Yaskawa INFORM job: A_ROOF_UPPER_0614_2_PAINT_34.JBI

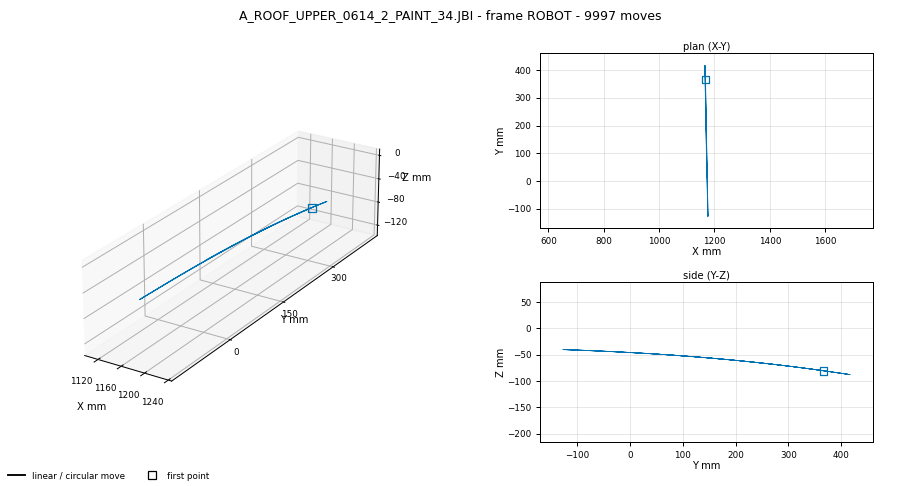
[picture p0: tool path of A_ROOF_UPPER_0614_2_PAINT_34.JBI in frame ROBOT, 9997 of 9997 moves have a stored position in this frame; points joined in program order, loops and branches not executed]
/JOB
//NAME A_ROOF_UPPER_0614_2_PAINT34
//POS
///NPOS 9997,0,0,0,0,0
///TOOL 1
///USER 0
///POSTYPE ROBOT
///RECTAN
///RCONF 1,0,0,0,0,0,0,0,0,0,0,0,0,0,0,0,0,0,0,0,0,0,0,0
C00000=1167.748,366.812,-80.185,-176.180,8.924,148.683
C00001=1167.752,366.565,-80.149,-176.183,8.920,148.683
C00002=1167.756,366.317,-80.115,-176.185,8.916,148.683
C00003=1167.761,366.035,-80.075,-176.187,8.912,148.682
C00004=1167.765,365.752,-80.035,-176.190,8.907,148.682
C00005=1167.770,365.471,-79.996,-176.191,8.904,148.681
C00006=1167.774,365.188,-79.956,-176.194,8.899,148.681
C00007=1167.778,364.940,-79.921,-176.196,8.895,148.680
C00008=1167.782,364.693,-79.887,-176.199,8.892,148.680
C00009=1167.786,364.446,-79.851,-176.200,8.888,148.680
C00010=1167.790,364.198,-79.817,-176.203,8.884,148.679
C00011=1167.794,363.950,-79.782,-176.205,8.880,148.679
C00012=1167.797,363.703,-79.747,-176.207,8.877,148.679
C00013=1167.802,363.456,-79.713,-176.209,8.872,148.678
C00014=1167.806,363.207,-79.678,-176.212,8.869,148.678
C00015=1167.809,362.960,-79.644,-176.214,8.865,148.677
C00016=1167.813,362.713,-79.608,-176.216,8.861,148.677
C00017=1167.818,362.465,-79.574,-176.218,8.858,148.677
C00018=1167.821,362.218,-79.540,-176.220,8.854,148.676
C00019=1167.825,361.970,-79.505,-176.223,8.850,148.676
C00020=1167.829,361.722,-79.470,-176.225,8.846,148.676
C00021=1167.833,361.475,-79.437,-176.227,8.843,148.675
C00022=1167.837,361.227,-79.402,-176.230,8.839,148.675
C00023=1167.842,360.980,-79.367,-176.232,8.835,148.675
C00024=1167.845,360.732,-79.332,-176.234,8.832,148.674
C00025=1167.849,360.485,-79.298,-176.237,8.828,148.674
C00026=1167.853,360.237,-79.263,-176.239,8.824,148.674
C00027=1167.857,359.990,-79.229,-176.241,8.820,148.673
C00028=1167.862,359.742,-79.195,-176.244,8.817,148.673
C00029=1167.865,359.494,-79.160,-176.245,8.813,148.673
C00030=1167.869,359.247,-79.126,-176.248,8.809,148.672
C00031=1167.873,358.999,-79.091,-176.251,8.806,148.672
C00032=1167.877,358.752,-79.057,-176.252,8.802,148.672
C00033=1167.881,358.504,-79.022,-176.255,8.798,148.671
C00034=1167.885,358.256,-78.989,-176.258,8.795,148.671
C00035=1167.890,358.009,-78.954,-176.259,8.791,148.671
C00036=1167.893,357.761,-78.920,-176.262,8.787,148.671
C00037=1167.897,357.514,-78.885,-176.265,8.784,148.670
C00038=1167.901,357.265,-78.852,-176.266,8.780,148.670
C00039=1167.906,357.018,-78.817,-176.269,8.776,148.670
C00040=1167.909,356.771,-78.784,-176.272,8.773,148.669
C00041=1167.913,356.523,-78.749,-176.274,8.769,148.669
C00042=1167.917,356.276,-78.715,-176.276,8.765,148.669
C00043=1167.921,356.027,-78.680,-176.279,8.762,148.669
C00044=1167.925,355.780,-78.646,-176.281,8.758,148.668
C00045=1167.930,355.532,-78.612,-176.283,8.754,148.668
C00046=1167.933,355.285,-78.578,-176.286,8.750,148.668
C00047=1167.938,355.037,-78.544,-176.288,8.747,148.667
C00048=1167.942,354.790,-78.510,-176.291,8.743,148.667
C00049=1167.945,354.542,-78.476,-176.293,8.739,148.667
C00050=1167.950,354.294,-78.442,-176.295,8.736,148.666
C00051=1167.953,354.047,-78.408,-176.298,8.732,148.666
C00052=1167.957,353.799,-78.373,-176.300,8.729,148.666
C00053=1167.962,353.551,-78.340,-176.302,8.725,148.666
C00054=1167.965,353.304,-78.306,-176.305,8.721,148.665
C00055=1167.969,353.056,-78.271,-176.307,8.718,148.665
C00056=1167.974,352.808,-78.238,-176.309,8.714,148.665
C00057=1167.978,352.561,-78.204,-176.312,8.711,148.665
C00058=1167.982,352.312,-78.170,-176.315,8.707,148.664
C00059=1167.985,352.065,-78.136,-176.316,8.703,148.664
C00060=1167.990,351.818,-78.102,-176.319,8.700,148.664
C00061=1167.994,351.570,-78.069,-176.322,8.696,148.664
C00062=1167.997,351.322,-78.034,-176.324,8.693,148.663
C00063=1168.002,351.074,-78.001,-176.326,8.689,148.663
C00064=1168.006,350.827,-77.967,-176.329,8.685,148.663
C00065=1168.010,350.579,-77.934,-176.331,8.682,148.662
C00066=1168.013,350.332,-77.899,-176.333,8.678,148.662
C00067=1168.018,350.084,-77.866,-176.335,8.675,148.662
C00068=1168.022,349.836,-77.832,-176.338,8.671,148.662
C00069=1168.026,349.589,-77.799,-176.341,8.668,148.661
C00070=1168.030,349.341,-77.764,-176.343,8.664,148.661
C00071=1168.034,349.093,-77.731,-176.346,8.660,148.661
C00072=1168.038,348.846,-77.697,-176.348,8.657,148.661
C00073=1168.042,348.598,-77.664,-176.350,8.654,148.661
C00074=1168.047,348.350,-77.630,-176.352,8.650,148.660
C00075=1168.050,348.102,-77.596,-176.355,8.646,148.660
C00076=1168.055,347.854,-77.562,-176.357,8.643,148.660
C00077=1168.059,347.607,-77.529,-176.360,8.639,148.659
C00078=1168.063,347.360,-77.495,-176.362,8.636,148.659
C00079=1168.067,347.112,-77.462,-176.365,8.632,148.659
C00080=1168.070,346.863,-77.429,-176.367,8.629,148.659
C00081=1168.075,346.616,-77.394,-176.369,8.625,148.659
C00082=1168.079,346.368,-77.361,-176.372,8.622,148.658
C00083=1168.083,346.121,-77.328,-176.374,8.618,148.658
C00084=1168.087,345.873,-77.294,-176.377,8.615,148.658
C00085=1168.091,345.626,-77.261,-176.379,8.611,148.658
C00086=1168.095,345.378,-77.228,-176.381,8.608,148.657
C00087=1168.099,345.130,-77.194,-176.384,8.604,148.657
C00088=1168.104,344.882,-77.161,-176.386,8.601,148.657
C00089=1168.107,344.634,-77.127,-176.389,8.597,148.657
C00090=1168.112,344.387,-77.093,-176.391,8.594,148.657
C00091=1168.116,344.139,-77.060,-176.394,8.590,148.656
C00092=1168.120,343.891,-77.027,-176.396,8.587,148.656
C00093=1168.124,343.644,-76.994,-176.398,8.583,148.656
C00094=1168.128,343.396,-76.961,-176.401,8.580,148.656
C00095=1168.132,343.148,-76.928,-176.404,8.576,148.655
C00096=1168.136,342.900,-76.895,-176.406,8.573,148.655
C00097=1168.140,342.653,-76.860,-176.408,8.569,148.655
C00098=1168.144,342.405,-76.827,-176.410,8.566,148.655
C00099=1168.148,342.157,-76.794,-176.413,8.562,148.655
C00100=1168.152,341.909,-76.761,-176.416,8.559,148.654
C00101=1168.156,341.662,-76.728,-176.418,8.555,148.654
C00102=1168.160,341.414,-76.695,-176.420,8.552,148.654
C00103=1168.164,341.166,-76.661,-176.423,8.549,148.654
C00104=1168.169,340.918,-76.628,-176.425,8.545,148.653
C00105=1168.173,340.671,-76.595,-176.428,8.542,148.653
C00106=1168.177,340.423,-76.562,-176.430,8.538,148.653
C00107=1168.182,340.143,-76.525,-176.433,8.534,148.653
C00108=1168.186,339.863,-76.488,-176.436,8.530,148.653
C00109=1168.191,339.585,-76.451,-176.438,8.527,148.652
C00110=1168.195,339.305,-76.413,-176.441,8.523,148.652
C00111=1168.200,339.057,-76.380,-176.444,8.519,148.652
C00112=1168.204,338.810,-76.347,-176.446,8.515,148.652
C00113=1168.208,338.562,-76.314,-176.449,8.512,148.652
C00114=1168.212,338.314,-76.281,-176.451,8.509,148.652
C00115=1168.216,338.066,-76.248,-176.454,8.506,148.651
C00116=1168.220,337.818,-76.216,-176.456,8.502,148.651
C00117=1168.224,337.571,-76.183,-176.459,8.498,148.651
C00118=1168.228,337.323,-76.150,-176.461,8.495,148.651
C00119=1168.232,337.075,-76.116,-176.463,8.492,148.650
C00120=1168.237,336.827,-76.084,-176.466,8.488,148.650
C00121=1168.240,336.579,-76.051,-176.468,8.485,148.650
C00122=1168.244,336.332,-76.018,-176.471,8.482,148.650
C00123=1168.249,336.083,-75.986,-176.474,8.478,148.650
C00124=1168.253,335.836,-75.953,-176.476,8.475,148.650
C00125=1168.257,335.588,-75.919,-176.478,8.471,148.649
C00126=1168.261,335.340,-75.888,-176.480,8.468,148.649
C00127=1168.265,335.092,-75.854,-176.483,8.465,148.649
C00128=1168.269,334.844,-75.821,-176.486,8.461,148.649
C00129=1168.273,334.596,-75.789,-176.488,8.458,148.649
C00130=1168.277,334.349,-75.756,-176.491,8.454,148.649
C00131=1168.282,334.102,-75.724,-176.493,8.451,148.648
C00132=1168.286,333.853,-75.691,-176.496,8.448,148.648
C00133=1168.289,333.606,-75.659,-176.498,8.445,148.648
C00134=1168.294,333.357,-75.626,-176.501,8.441,148.648
C00135=1168.298,333.110,-75.593,-176.503,8.437,148.648
C00136=1168.302,332.862,-75.561,-176.506,8.434,148.648
C00137=1168.306,332.614,-75.528,-176.508,8.431,148.647
C00138=1168.310,332.366,-75.495,-176.510,8.428,148.647
C00139=1168.314,332.118,-75.463,-176.513,8.424,148.647
C00140=1168.319,331.871,-75.431,-176.516,8.420,148.647
C00141=1168.323,331.623,-75.398,-176.518,8.417,148.647
C00142=1168.327,331.375,-75.366,-176.521,8.414,148.647
C00143=1168.331,331.127,-75.333,-176.523,8.411,148.646
C00144=1168.334,330.879,-75.301,-176.525,8.408,148.646
C00145=1168.339,330.631,-75.268,-176.528,8.405,148.646
C00146=1168.344,330.384,-75.236,-176.531,8.400,148.646
C00147=1168.347,330.136,-75.204,-176.533,8.397,148.646
C00148=1168.351,329.888,-75.171,-176.536,8.394,148.646
C00149=1168.355,329.640,-75.139,-176.538,8.391,148.646
C00150=1168.360,329.391,-75.106,-176.540,8.388,148.645
C00151=1168.364,329.144,-75.073,-176.543,8.384,148.645
C00152=1168.368,328.896,-75.042,-176.546,8.380,148.645
C00153=1168.372,328.648,-75.009,-176.548,8.377,148.645
C00154=1168.376,328.401,-74.977,-176.550,8.374,148.645
C00155=1168.380,328.152,-74.944,-176.553,8.371,148.645
C00156=1168.385,327.905,-74.913,-176.556,8.368,148.645
C00157=1168.389,327.657,-74.880,-176.558,8.364,148.644
C00158=1168.392,327.409,-74.848,-176.560,8.361,148.644
C00159=1168.397,327.161,-74.815,-176.563,8.357,148.644
C00160=1168.401,326.913,-74.783,-176.566,8.354,148.644
C00161=1168.405,326.665,-74.752,-176.568,8.351,148.644
C00162=1168.409,326.417,-74.720,-176.571,8.348,148.644
C00163=1168.413,326.170,-74.687,-176.573,8.344,148.643
C00164=1168.417,325.921,-74.655,-176.575,8.341,148.643
C00165=1168.422,325.674,-74.623,-176.578,8.338,148.643
C00166=1168.426,325.426,-74.591,-176.580,8.335,148.643
C00167=1168.430,325.178,-74.559,-176.583,8.331,148.643
C00168=1168.434,324.930,-74.527,-176.586,8.328,148.643
C00169=1168.438,324.682,-74.495,-176.588,8.324,148.643
C00170=1168.442,324.434,-74.463,-176.590,8.321,148.642
C00171=1168.447,324.186,-74.431,-176.593,8.318,148.642
C00172=1168.451,323.938,-74.399,-176.595,8.315,148.642
C00173=1168.455,323.690,-74.367,-176.598,8.312,148.642
C00174=1168.459,323.442,-74.335,-176.601,8.309,148.642
C00175=1168.463,323.194,-74.303,-176.603,8.304,148.642
C00176=1168.467,322.946,-74.272,-176.606,8.301,148.642
C00177=1168.471,322.698,-74.240,-176.608,8.298,148.642
C00178=1168.476,322.451,-74.208,-176.611,8.295,148.641
C00179=1168.479,322.203,-74.176,-176.613,8.292,148.641
C00180=1168.483,321.955,-74.144,-176.616,8.289,148.641
C00181=1168.488,321.707,-74.112,-176.618,8.286,148.641
C00182=1168.492,321.459,-74.080,-176.621,8.282,148.641
C00183=1168.496,321.211,-74.048,-176.623,8.279,148.641
C00184=1168.500,320.964,-74.017,-176.626,8.275,148.641
C00185=1168.504,320.715,-73.984,-176.629,8.272,148.641
C00186=1168.508,320.467,-73.952,-176.631,8.269,148.641
C00187=1168.513,320.219,-73.922,-176.634,8.266,148.640
C00188=1168.516,319.971,-73.890,-176.636,8.262,148.640
C00189=1168.521,319.724,-73.858,-176.639,8.259,148.640
C00190=1168.525,319.476,-73.826,-176.641,8.256,148.640
C00191=1168.529,319.227,-73.794,-176.644,8.253,148.640
C00192=1168.534,318.980,-73.763,-176.646,8.250,148.640
C00193=1168.537,318.731,-73.731,-176.649,8.247,148.640
C00194=1168.542,318.484,-73.700,-176.651,8.244,148.640
C00195=1168.546,318.236,-73.667,-176.654,8.239,148.639
C00196=1168.550,317.987,-73.636,-176.657,8.236,148.639
C00197=1168.554,317.740,-73.605,-176.659,8.233,148.639
C00198=1168.558,317.492,-73.573,-176.662,8.230,148.639
C00199=1168.563,317.244,-73.542,-176.664,8.227,148.639
C00200=1168.566,316.996,-73.510,-176.667,8.224,148.639
C00201=1168.571,316.748,-73.479,-176.669,8.221,148.639
C00202=1168.575,316.500,-73.448,-176.672,8.218,148.639
C00203=1168.580,316.252,-73.416,-176.674,8.214,148.639
C00204=1168.583,316.004,-73.384,-176.677,8.211,148.639
C00205=1168.587,315.755,-73.353,-176.679,8.208,148.639
C00206=1168.592,315.508,-73.321,-176.681,8.205,148.638
C00207=1168.596,315.259,-73.290,-176.685,8.201,148.638
C00208=1168.600,315.012,-73.259,-176.687,8.198,148.638
C00209=1168.604,314.763,-73.228,-176.690,8.195,148.638
C00210=1168.608,314.516,-73.196,-176.692,8.191,148.638
C00211=1168.613,314.239,-73.161,-176.695,8.188,148.638
C00212=1168.618,313.962,-73.127,-176.697,8.184,148.638
C00213=1168.622,313.685,-73.091,-176.700,8.181,148.638
C00214=1168.627,313.408,-73.056,-176.704,8.177,148.638
C00215=1168.632,313.160,-73.025,-176.706,8.174,148.638
C00216=1168.635,312.912,-72.993,-176.709,8.171,148.638
C00217=1168.640,312.664,-72.963,-176.711,8.168,148.637
C00218=1168.644,312.416,-72.931,-176.714,8.165,148.637
C00219=1168.648,312.168,-72.900,-176.716,8.162,148.637
C00220=1168.652,311.919,-72.869,-176.719,8.159,148.637
C00221=1168.657,311.672,-72.837,-176.721,8.155,148.637
C00222=1168.661,311.424,-72.807,-176.724,8.152,148.637
C00223=1168.664,311.176,-72.776,-176.726,8.149,148.637
C00224=1168.669,310.928,-72.745,-176.729,8.146,148.637
C00225=1168.673,310.680,-72.714,-176.731,8.143,148.637
C00226=1168.677,310.432,-72.683,-176.734,8.139,148.637
C00227=1168.682,310.184,-72.651,-176.737,8.136,148.636
C00228=1168.686,309.936,-72.620,-176.739,8.133,148.636
C00229=1168.690,309.688,-72.589,-176.742,8.129,148.636
C00230=1168.694,309.439,-72.558,-176.744,8.126,148.636
C00231=1168.699,309.192,-72.527,-176.747,8.123,148.636
C00232=1168.702,308.944,-72.497,-176.749,8.120,148.636
C00233=1168.707,308.695,-72.465,-176.752,8.117,148.636
C00234=1168.711,308.447,-72.435,-176.754,8.114,148.636
C00235=1168.716,308.199,-72.404,-176.757,8.111,148.636
C00236=1168.719,307.951,-72.372,-176.759,8.108,148.636
C00237=1168.723,307.704,-72.342,-176.762,8.105,148.636
C00238=1168.727,307.455,-72.311,-176.764,8.101,148.636
C00239=1168.732,307.207,-72.280,-176.767,8.098,148.636
C00240=1168.737,306.959,-72.249,-176.770,8.095,148.636
C00241=1168.741,306.710,-72.218,-176.772,8.092,148.635
C00242=1168.744,306.463,-72.188,-176.775,8.089,148.636
C00243=1168.749,306.215,-72.157,-176.777,8.086,148.635
C00244=1168.754,305.967,-72.126,-176.780,8.083,148.635
C00245=1168.757,305.719,-72.095,-176.783,8.080,148.635
C00246=1168.761,305.471,-72.064,-176.785,8.077,148.635
C00247=1168.766,305.223,-72.034,-176.788,8.074,148.635
C00248=1168.770,304.975,-72.003,-176.790,8.070,148.635
C00249=1168.774,304.727,-71.972,-176.793,8.067,148.635
C00250=1168.778,304.479,-71.942,-176.795,8.064,148.635
C00251=1168.783,304.230,-71.911,-176.798,8.061,148.635
C00252=1168.787,303.982,-71.880,-176.800,8.058,148.635
C00253=1168.791,303.734,-71.850,-176.803,8.055,148.635
C00254=1168.796,303.486,-71.820,-176.806,8.052,148.635
C00255=1168.800,303.238,-71.788,-176.808,8.049,148.635
C00256=1168.804,302.990,-71.758,-176.811,8.046,148.635
C00257=1168.808,302.742,-71.727,-176.813,8.043,148.635
C00258=1168.813,302.494,-71.697,-176.816,8.039,148.634
C00259=1168.816,302.246,-71.666,-176.818,8.036,148.634
C00260=1168.821,301.997,-71.636,-176.821,8.033,148.634
C00261=1168.825,301.749,-71.606,-176.823,8.030,148.634
C00262=1168.830,301.501,-71.575,-176.826,8.027,148.634
C00263=1168.834,301.253,-71.544,-176.829,8.024,148.634
C00264=1168.837,301.005,-71.514,-176.831,8.021,148.634
C00265=1168.842,300.757,-71.484,-176.834,8.018,148.634
C00266=1168.846,300.509,-71.454,-176.837,8.015,148.634
C00267=1168.851,300.261,-71.423,-176.839,8.012,148.634
C00268=1168.855,300.013,-71.393,-176.842,8.009,148.634
C00269=1168.859,299.764,-71.362,-176.844,8.006,148.634
C00270=1168.863,299.516,-71.332,-176.847,8.002,148.634
C00271=1168.868,299.268,-71.301,-176.849,7.999,148.634
C00272=1168.871,299.021,-71.271,-176.852,7.996,148.634
C00273=1168.876,298.772,-71.241,-176.854,7.993,148.634
C00274=1168.880,298.525,-71.211,-176.857,7.990,148.634
C00275=1168.884,298.276,-71.180,-176.860,7.987,148.634
C00276=1168.888,298.028,-71.150,-176.862,7.984,148.634
C00277=1168.893,297.780,-71.120,-176.865,7.981,148.634
C00278=1168.897,297.531,-71.090,-176.868,7.978,148.634
C00279=1168.902,297.283,-71.059,-176.870,7.975,148.634
C00280=1168.906,297.035,-71.030,-176.873,7.972,148.634
C00281=1168.911,296.787,-70.999,-176.875,7.969,148.634
C00282=1168.914,296.539,-70.969,-176.878,7.965,148.633
C00283=1168.918,296.291,-70.939,-176.880,7.962,148.633
C00284=1168.923,296.043,-70.908,-176.883,7.959,148.633
C00285=1168.927,295.794,-70.879,-176.885,7.956,148.633
C00286=1168.931,295.547,-70.849,-176.888,7.953,148.633
C00287=1168.936,295.298,-70.819,-176.891,7.950,148.633
C00288=1168.940,295.050,-70.789,-176.894,7.947,148.633
C00289=1168.944,294.802,-70.759,-176.896,7.944,148.633
C00290=1168.948,294.554,-70.728,-176.899,7.941,148.633
C00291=1168.952,294.305,-70.699,-176.901,7.938,148.633
C00292=1168.956,294.057,-70.669,-176.904,7.935,148.633
C00293=1168.961,293.809,-70.638,-176.907,7.932,148.633
C00294=1168.965,293.561,-70.609,-176.909,7.929,148.633
C00295=1168.969,293.313,-70.579,-176.912,7.926,148.633
C00296=1168.974,293.065,-70.549,-176.914,7.922,148.633
C00297=1168.978,292.816,-70.519,-176.917,7.919,148.633
C00298=1168.982,292.569,-70.489,-176.920,7.917,148.633
C00299=1168.987,292.320,-70.459,-176.922,7.913,148.633
C00300=1168.991,292.072,-70.430,-176.924,7.911,148.633
C00301=1168.995,291.824,-70.399,-176.927,7.908,148.633
C00302=1168.999,291.576,-70.370,-176.930,7.905,148.633
C00303=1169.004,291.327,-70.340,-176.932,7.902,148.633
C00304=1169.008,291.079,-70.310,-176.935,7.899,148.633
C00305=1169.012,290.831,-70.280,-176.937,7.896,148.633
C00306=1169.016,290.583,-70.251,-176.940,7.893,148.633
C00307=1169.020,290.335,-70.221,-176.943,7.890,148.633
C00308=1169.025,290.086,-70.191,-176.945,7.887,148.633
C00309=1169.029,289.838,-70.162,-176.948,7.884,148.633
C00310=1169.033,289.590,-70.132,-176.951,7.881,148.633
C00311=1169.037,289.342,-70.102,-176.953,7.877,148.633
C00312=1169.042,289.094,-70.073,-176.956,7.874,148.633
C00313=1169.046,288.846,-70.043,-176.959,7.871,148.633
C00314=1169.051,288.597,-70.013,-176.961,7.869,148.633
C00315=1169.055,288.323,-69.981,-176.964,7.866,148.633
C00316=1169.060,288.047,-69.948,-176.967,7.863,148.633
C00317=1169.065,287.773,-69.915,-176.970,7.858,148.633
C00318=1169.070,287.498,-69.882,-176.972,7.855,148.633
C00319=1169.074,287.249,-69.853,-176.975,7.853,148.633
C00320=1169.078,287.001,-69.823,-176.978,7.850,148.633
C00321=1169.082,286.753,-69.794,-176.981,7.847,148.633
C00322=1169.086,286.505,-69.765,-176.983,7.843,148.633
C00323=1169.091,286.256,-69.735,-176.986,7.840,148.633
C00324=1169.095,286.008,-69.706,-176.988,7.837,148.633
C00325=1169.099,285.760,-69.676,-176.991,7.835,148.633
C00326=1169.104,285.512,-69.647,-176.993,7.832,148.633
C00327=1169.108,285.264,-69.618,-176.996,7.829,148.633
C00328=1169.112,285.016,-69.588,-176.998,7.826,148.633
C00329=1169.116,284.767,-69.559,-177.001,7.823,148.633
C00330=1169.120,284.519,-69.529,-177.004,7.820,148.633
C00331=1169.125,284.271,-69.500,-177.007,7.817,148.633
C00332=1169.129,284.022,-69.471,-177.009,7.814,148.633
C00333=1169.133,283.774,-69.442,-177.012,7.811,148.633
C00334=1169.138,283.526,-69.413,-177.014,7.808,148.633
C00335=1169.142,283.278,-69.383,-177.017,7.805,148.633
C00336=1169.146,283.030,-69.354,-177.019,7.803,148.633
C00337=1169.151,282.781,-69.324,-177.022,7.800,148.633
C00338=1169.155,282.533,-69.295,-177.025,7.797,148.633
C00339=1169.160,282.285,-69.266,-177.027,7.793,148.633
C00340=1169.164,282.037,-69.237,-177.030,7.790,148.633
C00341=1169.168,281.788,-69.208,-177.033,7.788,148.633
C00342=1169.172,281.540,-69.178,-177.035,7.785,148.633
C00343=1169.177,281.291,-69.149,-177.038,7.782,148.633
C00344=1169.180,281.043,-69.120,-177.041,7.779,148.633
C00345=1169.185,280.796,-69.091,-177.043,7.775,148.633
C00346=1169.190,280.547,-69.063,-177.045,7.773,148.633
C00347=1169.194,280.299,-69.033,-177.048,7.770,148.633
C00348=1169.198,280.050,-69.004,-177.051,7.767,148.633
C00349=1169.203,279.802,-68.975,-177.053,7.764,148.633
C00350=1169.207,279.554,-68.946,-177.056,7.761,148.633
C00351=1169.211,279.306,-68.917,-177.059,7.758,148.633
C00352=1169.215,279.057,-68.888,-177.062,7.755,148.633
C00353=1169.220,278.809,-68.859,-177.064,7.752,148.633
C00354=1169.225,278.561,-68.830,-177.066,7.750,148.633
C00355=1169.229,278.312,-68.801,-177.069,7.747,148.633
C00356=1169.232,278.064,-68.772,-177.072,7.744,148.633
C00357=1169.237,277.816,-68.744,-177.074,7.741,148.633
C00358=1169.241,277.568,-68.714,-177.077,7.738,148.633
C00359=1169.246,277.319,-68.686,-177.080,7.735,148.633
C00360=1169.249,277.071,-68.657,-177.083,7.732,148.633
C00361=1169.254,276.823,-68.628,-177.085,7.729,148.633
C00362=1169.259,276.575,-68.599,-177.087,7.727,148.633
C00363=1169.262,276.326,-68.571,-177.090,7.724,148.633
C00364=1169.267,276.078,-68.542,-177.093,7.721,148.633
C00365=1169.272,275.830,-68.513,-177.095,7.718,148.633
C00366=1169.276,275.581,-68.484,-177.098,7.715,148.633
C00367=1169.280,275.333,-68.455,-177.101,7.712,148.633
C00368=1169.285,275.085,-68.427,-177.104,7.709,148.633
C00369=1169.289,274.836,-68.398,-177.106,7.707,148.633
C00370=1169.293,274.588,-68.369,-177.108,7.704,148.634
C00371=1169.298,274.340,-68.341,-177.111,7.701,148.634
C00372=1169.302,274.091,-68.312,-177.114,7.698,148.634
C00373=1169.306,273.843,-68.283,-177.117,7.695,148.634
C00374=1169.311,273.594,-68.255,-177.119,7.692,148.633
C00375=1169.314,273.347,-68.226,-177.122,7.689,148.634
C00376=1169.319,273.098,-68.198,-177.124,7.686,148.634
C00377=1169.324,272.849,-68.169,-177.127,7.683,148.634
C00378=1169.327,272.601,-68.140,-177.129,7.681,148.634
C00379=1169.332,272.353,-68.112,-177.132,7.678,148.634
C00380=1169.336,272.105,-68.084,-177.135,7.675,148.634
C00381=1169.340,271.856,-68.055,-177.138,7.672,148.634
C00382=1169.345,271.608,-68.026,-177.140,7.669,148.634
C00383=1169.349,271.360,-67.998,-177.143,7.667,148.634
C00384=1169.354,271.112,-67.969,-177.145,7.664,148.634
C00385=1169.358,270.863,-67.941,-177.148,7.661,148.634
C00386=1169.363,270.615,-67.913,-177.151,7.658,148.634
C00387=1169.367,270.366,-67.885,-177.154,7.655,148.634
C00388=1169.371,270.118,-67.855,-177.156,7.653,148.634
C00389=1169.375,269.870,-67.827,-177.159,7.650,148.634
C00390=1169.380,269.621,-67.799,-177.161,7.647,148.634
C00391=1169.384,269.373,-67.771,-177.164,7.644,148.634
C00392=1169.389,269.124,-67.742,-177.167,7.641,148.634
C00393=1169.393,268.877,-67.714,-177.169,7.638,148.635
C00394=1169.397,268.628,-67.686,-177.172,7.636,148.635
C00395=1169.402,268.380,-67.658,-177.174,7.633,148.635
C00396=1169.405,268.131,-67.630,-177.177,7.630,148.635
C00397=1169.410,267.882,-67.601,-177.180,7.627,148.635
C00398=1169.414,267.634,-67.573,-177.183,7.624,148.635
C00399=1169.419,267.386,-67.545,-177.185,7.622,148.635
C00400=1169.423,267.138,-67.517,-177.188,7.619,148.635
C00401=1169.428,266.889,-67.488,-177.190,7.616,148.635
C00402=1169.432,266.641,-67.460,-177.193,7.613,148.635
C00403=1169.436,266.392,-67.432,-177.196,7.610,148.635
C00404=1169.441,266.144,-67.404,-177.198,7.608,148.635
C00405=1169.445,265.896,-67.376,-177.201,7.605,148.635
C00406=1169.450,265.647,-67.347,-177.204,7.602,148.635
C00407=1169.454,265.399,-67.319,-177.206,7.599,148.635
C00408=1169.458,265.151,-67.291,-177.209,7.596,148.635
C00409=1169.463,264.903,-67.263,-177.211,7.594,148.635
C00410=1169.467,264.654,-67.235,-177.214,7.591,148.636
C00411=1169.471,264.406,-67.208,-177.217,7.588,148.636
C00412=1169.476,264.157,-67.179,-177.219,7.585,148.636
C00413=1169.480,263.909,-67.151,-177.222,7.582,148.636
C00414=1169.484,263.660,-67.123,-177.224,7.580,148.636
C00415=1169.489,263.412,-67.096,-177.227,7.577,148.636
C00416=1169.494,263.164,-67.068,-177.230,7.574,148.636
C00417=1169.497,262.915,-67.039,-177.233,7.571,148.636
C00418=1169.502,262.667,-67.012,-177.235,7.569,148.636
C00419=1169.506,262.394,-66.981,-177.238,7.565,148.636
C00420=1169.511,262.121,-66.950,-177.241,7.562,148.636
C00421=1169.516,261.848,-66.920,-177.244,7.559,148.636
C00422=1169.521,261.575,-66.889,-177.247,7.556,148.636
C00423=1169.525,261.326,-66.861,-177.250,7.553,148.636
C00424=1169.530,261.077,-66.834,-177.252,7.550,148.637
C00425=1169.534,260.829,-66.806,-177.255,7.548,148.637
C00426=1169.538,260.581,-66.778,-177.257,7.545,148.637
C00427=1169.543,260.332,-66.751,-177.260,7.542,148.637
C00428=1169.547,260.084,-66.723,-177.263,7.539,148.637
C00429=1169.551,259.835,-66.695,-177.265,7.537,148.637
C00430=1169.556,259.587,-66.667,-177.268,7.534,148.637
C00431=1169.560,259.338,-66.639,-177.271,7.531,148.637
C00432=1169.565,259.090,-66.612,-177.274,7.529,148.637
C00433=1169.569,258.842,-66.584,-177.276,7.526,148.637
C00434=1169.573,258.593,-66.557,-177.279,7.523,148.637
C00435=1169.578,258.345,-66.529,-177.281,7.520,148.637
C00436=1169.582,258.096,-66.502,-177.284,7.517,148.638
C00437=1169.587,257.849,-66.474,-177.286,7.515,148.638
C00438=1169.591,257.599,-66.446,-177.289,7.512,148.638
C00439=1169.596,257.351,-66.418,-177.292,7.509,148.638
C00440=1169.600,257.103,-66.391,-177.295,7.506,148.638
C00441=1169.604,256.854,-66.363,-177.297,7.505,148.638
C00442=1169.609,256.606,-66.336,-177.300,7.502,148.638
C00443=1169.613,256.358,-66.308,-177.303,7.499,148.638
C00444=1169.617,256.109,-66.281,-177.306,7.496,148.638
C00445=1169.622,255.860,-66.254,-177.308,7.494,148.638
C00446=1169.626,255.612,-66.226,-177.310,7.491,148.638
C00447=1169.631,255.364,-66.199,-177.313,7.488,148.639
C00448=1169.635,255.115,-66.171,-177.316,7.485,148.639
C00449=1169.639,254.867,-66.144,-177.319,7.483,148.639
C00450=1169.644,254.618,-66.117,-177.321,7.480,148.639
C00451=1169.648,254.370,-66.089,-177.324,7.477,148.639
C00452=1169.652,254.121,-66.061,-177.326,7.475,148.639
C00453=1169.657,253.873,-66.034,-177.329,7.472,148.639
C00454=1169.662,253.624,-66.007,-177.332,7.469,148.639
C00455=1169.666,253.376,-65.979,-177.335,7.466,148.639
C00456=1169.671,253.128,-65.952,-177.337,7.464,148.640
C00457=1169.675,252.878,-65.925,-177.340,7.461,148.640
C00458=1169.679,252.630,-65.898,-177.343,7.458,148.640
C00459=1169.683,252.382,-65.871,-177.345,7.456,148.640
C00460=1169.688,252.134,-65.844,-177.348,7.453,148.640
C00461=1169.692,251.885,-65.816,-177.350,7.450,148.640
C00462=1169.696,251.636,-65.789,-177.354,7.448,148.640
C00463=1169.701,251.388,-65.762,-177.356,7.445,148.640
C00464=1169.705,251.140,-65.734,-177.359,7.442,148.640
C00465=1169.710,250.891,-65.707,-177.361,7.440,148.640
C00466=1169.714,250.643,-65.681,-177.363,7.437,148.641
C00467=1169.718,250.394,-65.653,-177.366,7.434,148.641
C00468=1169.723,250.145,-65.626,-177.369,7.432,148.641
C00469=1169.727,249.897,-65.599,-177.372,7.430,148.641
C00470=1169.732,249.648,-65.572,-177.374,7.427,148.641
C00471=1169.737,249.400,-65.545,-177.377,7.424,148.641
C00472=1169.740,249.152,-65.519,-177.380,7.421,148.641
C00473=1169.745,248.903,-65.492,-177.383,7.419,148.641
C00474=1169.749,248.654,-65.464,-177.385,7.416,148.642
C00475=1169.754,248.406,-65.437,-177.388,7.413,148.642
C00476=1169.759,248.157,-65.410,-177.390,7.411,148.642
C00477=1169.762,247.909,-65.384,-177.393,7.408,148.642
C00478=1169.767,247.660,-65.357,-177.396,7.405,148.642
C00479=1169.772,247.412,-65.329,-177.398,7.403,148.642
C00480=1169.776,247.163,-65.302,-177.401,7.400,148.642
C00481=1169.780,246.915,-65.276,-177.404,7.397,148.642
C00482=1169.785,246.667,-65.249,-177.407,7.395,148.643
C00483=1169.790,246.418,-65.222,-177.409,7.393,148.643
C00484=1169.793,246.169,-65.195,-177.412,7.390,148.643
C00485=1169.798,245.921,-65.168,-177.414,7.387,148.643
C00486=1169.802,245.672,-65.141,-177.417,7.384,148.643
C00487=1169.806,245.424,-65.114,-177.420,7.382,148.643
C00488=1169.811,245.175,-65.088,-177.422,7.380,148.643
C00489=1169.816,244.927,-65.061,-177.425,7.377,148.643
C00490=1169.820,244.678,-65.035,-177.428,7.374,148.643
C00491=1169.824,244.430,-65.007,-177.431,7.372,148.644
C00492=1169.829,244.181,-64.980,-177.433,7.369,148.644
C00493=1169.833,243.933,-64.955,-177.436,7.366,148.644
C00494=1169.838,243.684,-64.928,-177.438,7.364,148.644
C00495=1169.843,243.436,-64.901,-177.441,7.361,148.644
C00496=1169.846,243.187,-64.874,-177.444,7.358,148.644
C00497=1169.851,242.938,-64.848,-177.446,7.356,148.644
C00498=1169.855,242.690,-64.821,-177.450,7.354,148.645
C00499=1169.860,242.442,-64.794,-177.452,7.351,148.645
C00500=1169.864,242.193,-64.768,-177.455,7.348,148.645
C00501=1169.869,241.944,-64.741,-177.457,7.346,148.645
C00502=1169.874,241.696,-64.714,-177.460,7.344,148.645
C00503=1169.877,241.448,-64.688,-177.463,7.341,148.645
C00504=1169.882,241.199,-64.661,-177.466,7.338,148.645
C00505=1169.886,240.950,-64.635,-177.468,7.336,148.646
C00506=1169.891,240.702,-64.608,-177.471,7.333,148.646
C00507=1169.895,240.453,-64.582,-177.474,7.330,148.646
C00508=1169.900,240.205,-64.555,-177.476,7.328,148.646
C00509=1169.904,239.956,-64.529,-177.479,7.325,148.646
C00510=1169.909,239.707,-64.502,-177.481,7.323,148.646
C00511=1169.913,239.458,-64.477,-177.484,7.320,148.646
C00512=1169.918,239.210,-64.450,-177.487,7.318,148.647
C00513=1169.922,238.962,-64.424,-177.489,7.316,148.647
C00514=1169.927,238.713,-64.397,-177.492,7.313,148.647
C00515=1169.931,238.465,-64.371,-177.495,7.310,148.647
C00516=1169.935,238.216,-64.345,-177.498,7.308,148.647
C00517=1169.940,237.967,-64.319,-177.500,7.305,148.647
C00518=1169.944,237.719,-64.292,-177.503,7.303,148.648
C00519=1169.949,237.470,-64.266,-177.506,7.300,148.648
C00520=1169.953,237.222,-64.239,-177.509,7.297,148.648
C00521=1169.957,236.973,-64.213,-177.511,7.295,148.648
C00522=1169.962,236.724,-64.186,-177.514,7.292,148.648
C00523=1169.967,236.453,-64.158,-177.517,7.289,148.648
C00524=1169.972,236.182,-64.129,-177.520,7.287,148.649
C00525=1169.977,235.910,-64.101,-177.523,7.284,148.649
C00526=1169.981,235.639,-64.073,-177.526,7.281,148.649
C00527=1169.986,235.389,-64.046,-177.528,7.279,148.649
C00528=1169.990,235.141,-64.020,-177.531,7.276,148.649
C00529=1169.995,234.892,-63.994,-177.534,7.274,148.650
C00530=1170.000,234.643,-63.968,-177.536,7.271,148.650
C00531=1170.004,234.395,-63.942,-177.538,7.269,148.650
C00532=1170.008,234.147,-63.916,-177.542,7.267,148.650
C00533=1170.013,233.898,-63.889,-177.544,7.264,148.650
C00534=1170.017,233.649,-63.864,-177.547,7.262,148.650
C00535=1170.021,233.401,-63.837,-177.550,7.259,148.650
C00536=1170.026,233.152,-63.812,-177.552,7.257,148.651
C00537=1170.031,232.904,-63.786,-177.555,7.254,148.651
C00538=1170.035,232.655,-63.760,-177.557,7.252,148.651
C00539=1170.040,232.406,-63.734,-177.560,7.249,148.651
C00540=1170.044,232.158,-63.708,-177.563,7.246,148.651
C00541=1170.048,231.909,-63.681,-177.566,7.244,148.651
C00542=1170.053,231.661,-63.656,-177.569,7.242,148.652
C00543=1170.058,231.412,-63.630,-177.571,7.240,148.652
C00544=1170.062,231.163,-63.604,-177.574,7.237,148.652
C00545=1170.067,230.914,-63.578,-177.577,7.235,148.652
C00546=1170.071,230.666,-63.552,-177.579,7.232,148.652
C00547=1170.075,230.418,-63.526,-177.582,7.229,148.653
C00548=1170.080,230.169,-63.500,-177.585,7.227,148.653
C00549=1170.084,229.920,-63.475,-177.587,7.224,148.653
C00550=1170.089,229.672,-63.449,-177.590,7.222,148.653
C00551=1170.093,229.423,-63.424,-177.593,7.219,148.653
C00552=1170.098,229.174,-63.397,-177.596,7.218,148.654
C00553=1170.102,228.925,-63.371,-177.598,7.215,148.654
C00554=1170.107,228.677,-63.346,-177.600,7.213,148.654
C00555=1170.111,228.428,-63.320,-177.604,7.210,148.654
C00556=1170.115,228.180,-63.295,-177.606,7.208,148.654
C00557=1170.120,227.931,-63.269,-177.609,7.205,148.654
C00558=1170.124,227.683,-63.243,-177.611,7.203,148.655
C00559=1170.129,227.434,-63.218,-177.615,7.200,148.655
C00560=1170.134,227.186,-63.192,-177.617,7.198,148.655
C00561=1170.138,226.937,-63.167,-177.619,7.195,148.655
C00562=1170.143,226.688,-63.140,-177.623,7.193,148.655
C00563=1170.148,226.440,-63.115,-177.625,7.191,148.655
C00564=1170.152,226.190,-63.090,-177.628,7.188,148.656
C00565=1170.156,225.941,-63.064,-177.630,7.186,148.656
C00566=1170.161,225.693,-63.039,-177.634,7.183,148.656
C00567=1170.165,225.445,-63.013,-177.636,7.181,148.656
C00568=1170.170,225.196,-62.987,-177.639,7.179,148.657
C00569=1170.174,224.948,-62.962,-177.641,7.176,148.657
C00570=1170.179,224.699,-62.936,-177.644,7.173,148.657
C00571=1170.183,224.449,-62.911,-177.647,7.172,148.657
C00572=1170.188,224.201,-62.886,-177.649,7.169,148.657
C00573=1170.192,223.952,-62.860,-177.652,7.167,148.658
C00574=1170.197,223.704,-62.834,-177.655,7.164,148.658
C00575=1170.201,223.455,-62.810,-177.657,7.162,148.658
C00576=1170.205,223.206,-62.784,-177.660,7.159,148.658
C00577=1170.210,222.958,-62.759,-177.663,7.157,148.658
C00578=1170.214,222.710,-62.733,-177.666,7.154,148.658
C00579=1170.219,222.461,-62.708,-177.668,7.153,148.659
C00580=1170.223,222.212,-62.683,-177.671,7.150,148.659
C00581=1170.228,221.963,-62.657,-177.674,7.148,148.659
C00582=1170.233,221.714,-62.632,-177.676,7.145,148.659
C00583=1170.237,221.466,-62.606,-177.679,7.143,148.660
C00584=1170.242,221.218,-62.581,-177.682,7.140,148.660
C00585=1170.246,220.968,-62.556,-177.685,7.138,148.660
C00586=1170.250,220.720,-62.531,-177.687,7.136,148.660
C00587=1170.255,220.472,-62.506,-177.690,7.134,148.660
C00588=1170.259,220.222,-62.480,-177.693,7.131,148.661
C00589=1170.264,219.974,-62.455,-177.695,7.129,148.661
C00590=1170.269,219.725,-62.430,-177.698,7.126,148.661
C00591=1170.273,219.477,-62.405,-177.701,7.124,148.661
C00592=1170.277,219.227,-62.380,-177.704,7.121,148.661
C00593=1170.282,218.979,-62.355,-177.706,7.120,148.662
C00594=1170.287,218.730,-62.330,-177.708,7.117,148.662
C00595=1170.291,218.482,-62.304,-177.712,7.115,148.662
C00596=1170.295,218.233,-62.280,-177.714,7.113,148.662
C00597=1170.300,217.985,-62.255,-177.717,7.110,148.663
C00598=1170.305,217.735,-62.230,-177.719,7.108,148.663
C00599=1170.309,217.487,-62.204,-177.723,7.105,148.663
C00600=1170.313,217.238,-62.180,-177.725,7.103,148.663
C00601=1170.318,216.990,-62.154,-177.728,7.101,148.663
C00602=1170.323,216.740,-62.129,-177.730,7.098,148.664
C00603=1170.327,216.492,-62.104,-177.733,7.096,148.664
C00604=1170.331,216.243,-62.080,-177.736,7.094,148.664
C00605=1170.336,215.994,-62.055,-177.738,7.092,148.664
C00606=1170.340,215.746,-62.029,-177.742,7.089,148.665
C00607=1170.345,215.497,-62.005,-177.744,7.087,148.665
C00608=1170.350,215.249,-61.980,-177.747,7.085,148.665
C00609=1170.354,215.000,-61.955,-177.749,7.082,148.665
C00610=1170.359,214.751,-61.931,-177.752,7.080,148.665
C00611=1170.363,214.502,-61.905,-177.755,7.078,148.666
C00612=1170.368,214.254,-61.880,-177.757,7.076,148.666
C00613=1170.372,214.005,-61.856,-177.760,7.073,148.666
C00614=1170.377,213.756,-61.831,-177.763,7.071,148.666
C00615=1170.382,213.508,-61.806,-177.765,7.068,148.666
C00616=1170.386,213.259,-61.781,-177.768,7.066,148.667
C00617=1170.391,213.010,-61.756,-177.771,7.064,148.667
C00618=1170.394,212.761,-61.732,-177.774,7.062,148.667
C00619=1170.399,212.513,-61.707,-177.776,7.060,148.668
C00620=1170.404,212.264,-61.682,-177.779,7.057,148.668
C00621=1170.408,212.015,-61.658,-177.782,7.055,148.668
C00622=1170.413,211.766,-61.633,-177.784,7.052,148.668
C00623=1170.417,211.517,-61.608,-177.787,7.050,148.668
C00624=1170.422,211.269,-61.583,-177.790,7.048,148.669
C00625=1170.426,211.021,-61.559,-177.792,7.046,148.669
C00626=1170.431,210.771,-61.534,-177.795,7.044,148.669
C00627=1170.436,210.501,-61.507,-177.798,7.041,148.669
C00628=1170.441,210.231,-61.481,-177.801,7.038,148.670
C00629=1170.446,209.959,-61.454,-177.804,7.037,148.670
C00630=1170.451,209.689,-61.427,-177.807,7.034,148.670
C00631=1170.456,209.441,-61.403,-177.810,7.031,148.670
C00632=1170.460,209.191,-61.378,-177.813,7.029,148.671
C00633=1170.465,208.943,-61.354,-177.815,7.027,148.671
C00634=1170.469,208.695,-61.329,-177.818,7.025,148.671
C00635=1170.473,208.446,-61.304,-177.821,7.023,148.671
C00636=1170.478,208.197,-61.280,-177.823,7.020,148.672
C00637=1170.483,207.949,-61.256,-177.826,7.018,148.672
C00638=1170.488,207.700,-61.231,-177.828,7.016,148.672
C00639=1170.492,207.450,-61.207,-177.831,7.013,148.672
C00640=1170.496,207.202,-61.183,-177.834,7.012,148.673
C00641=1170.501,206.953,-61.159,-177.836,7.009,148.673
C00642=1170.505,206.704,-61.134,-177.840,7.007,148.673
C00643=1170.510,206.455,-61.109,-177.842,7.005,148.673
C00644=1170.515,206.207,-61.085,-177.845,7.002,148.674
C00645=1170.519,205.958,-61.061,-177.848,7.000,148.674
C00646=1170.524,205.709,-61.036,-177.850,6.998,148.674
C00647=1170.528,205.460,-61.012,-177.853,6.996,148.674
C00648=1170.533,205.212,-60.988,-177.856,6.994,148.675
C00649=1170.538,204.963,-60.963,-177.858,6.992,148.675
C00650=1170.542,204.714,-60.940,-177.861,6.989,148.675
C00651=1170.547,204.465,-60.915,-177.863,6.987,148.675
C00652=1170.551,204.216,-60.891,-177.866,6.985,148.676
C00653=1170.556,203.968,-60.867,-177.869,6.983,148.676
C00654=1170.561,203.719,-60.842,-177.872,6.980,148.676
C00655=1170.565,203.470,-60.819,-177.875,6.978,148.676
C00656=1170.569,203.221,-60.794,-177.877,6.976,148.677
C00657=1170.574,202.973,-60.770,-177.880,6.974,148.677
C00658=1170.579,202.724,-60.746,-177.883,6.971,148.677
C00659=1170.583,202.475,-60.722,-177.886,6.970,148.678
C00660=1170.587,202.226,-60.698,-177.888,6.967,148.678
C00661=1170.592,201.977,-60.674,-177.891,6.965,148.678
C00662=1170.597,201.729,-60.649,-177.894,6.963,148.678
C00663=1170.601,201.480,-60.626,-177.896,6.961,148.678
C00664=1170.606,201.231,-60.602,-177.899,6.958,148.679
C00665=1170.610,200.983,-60.578,-177.901,6.956,148.679
C00666=1170.615,200.733,-60.553,-177.904,6.954,148.679
C00667=1170.619,200.484,-60.529,-177.907,6.952,148.680
C00668=1170.624,200.235,-60.506,-177.909,6.950,148.680
C00669=1170.629,199.987,-60.482,-177.912,6.948,148.680
C00670=1170.633,199.739,-60.458,-177.915,6.945,148.680
C00671=1170.638,199.490,-60.434,-177.918,6.944,148.681
C00672=1170.643,199.241,-60.410,-177.920,6.941,148.681
C00673=1170.647,198.991,-60.386,-177.923,6.939,148.681
C00674=1170.651,198.743,-60.362,-177.926,6.937,148.681
C00675=1170.656,198.494,-60.338,-177.928,6.935,148.682
C00676=1170.660,198.245,-60.314,-177.932,6.932,148.682
C00677=1170.665,197.997,-60.290,-177.934,6.931,148.682
C00678=1170.669,197.748,-60.267,-177.936,6.928,148.682
C00679=1170.675,197.499,-60.242,-177.940,6.926,148.683
C00680=1170.679,197.250,-60.219,-177.942,6.924,148.683
C00681=1170.684,197.002,-60.195,-177.945,6.922,148.683
C00682=1170.688,196.753,-60.172,-177.947,6.920,148.684
C00683=1170.693,196.503,-60.148,-177.951,6.918,148.684
C00684=1170.697,196.254,-60.124,-177.953,6.915,148.684
C00685=1170.702,196.005,-60.100,-177.955,6.914,148.684
C00686=1170.706,195.757,-60.076,-177.959,6.911,148.685
C00687=1170.711,195.508,-60.053,-177.961,6.909,148.685
C00688=1170.715,195.260,-60.029,-177.963,6.907,148.685
C00689=1170.720,195.011,-60.006,-177.967,6.905,148.686
C00690=1170.724,194.761,-59.982,-177.969,6.903,148.686
C00691=1170.729,194.513,-59.958,-177.972,6.901,148.686
C00692=1170.734,194.264,-59.935,-177.974,6.899,148.686
C00693=1170.738,194.015,-59.911,-177.978,6.896,148.687
C00694=1170.743,193.767,-59.887,-177.980,6.895,148.687
C00695=1170.747,193.518,-59.864,-177.982,6.892,148.687
C00696=1170.752,193.269,-59.841,-177.986,6.890,148.687
C00697=1170.757,193.019,-59.817,-177.988,6.888,148.688
C00698=1170.761,192.771,-59.793,-177.991,6.886,148.688
C00699=1170.766,192.522,-59.770,-177.993,6.884,148.688
C00700=1170.771,192.273,-59.746,-177.996,6.882,148.689
C00701=1170.775,192.024,-59.723,-177.999,6.880,148.689
C00702=1170.780,191.776,-59.699,-178.001,6.878,148.689
C00703=1170.784,191.527,-59.676,-178.004,6.876,148.689
C00704=1170.789,191.277,-59.652,-178.007,6.873,148.690
C00705=1170.794,191.028,-59.629,-178.010,6.872,148.690
C00706=1170.798,190.779,-59.606,-178.012,6.869,148.690
C00707=1170.803,190.531,-59.582,-178.015,6.867,148.691
C00708=1170.807,190.282,-59.559,-178.018,6.865,148.691
C00709=1170.812,190.034,-59.536,-178.021,6.863,148.691
C00710=1170.817,189.785,-59.512,-178.023,6.861,148.691
C00711=1170.822,189.536,-59.489,-178.026,6.859,148.692
C00712=1170.826,189.287,-59.466,-178.029,6.857,148.692
C00713=1170.831,189.038,-59.442,-178.032,6.855,148.693
C00714=1170.836,188.789,-59.419,-178.034,6.853,148.693
C00715=1170.839,188.541,-59.395,-178.037,6.850,148.693
C00716=1170.844,188.292,-59.372,-178.040,6.849,148.693
C00717=1170.849,188.043,-59.349,-178.042,6.847,148.694
C00718=1170.853,187.794,-59.325,-178.045,6.845,148.694
C00719=1170.858,187.545,-59.302,-178.048,6.842,148.694
C00720=1170.863,187.296,-59.279,-178.050,6.840,148.695
C00721=1170.867,187.048,-59.256,-178.053,6.839,148.695
C00722=1170.872,186.798,-59.233,-178.055,6.836,148.695
C00723=1170.877,186.549,-59.210,-178.058,6.835,148.695
C00724=1170.881,186.300,-59.186,-178.061,6.832,148.696
C00725=1170.885,186.052,-59.163,-178.064,6.830,148.696
C00726=1170.890,185.803,-59.140,-178.067,6.829,148.696
C00727=1170.895,185.553,-59.117,-178.069,6.826,148.697
C00728=1170.900,185.305,-59.094,-178.072,6.824,148.697
C00729=1170.904,185.056,-59.072,-178.075,6.822,148.697
C00730=1170.909,184.807,-59.048,-178.077,6.820,148.698
C00731=1170.914,184.537,-59.023,-178.081,6.818,148.698
C00732=1170.919,184.268,-58.999,-178.083,6.816,148.698
C00733=1170.924,183.999,-58.973,-178.087,6.813,148.699
C00734=1170.929,183.729,-58.948,-178.089,6.811,148.699
C00735=1170.933,183.480,-58.925,-178.092,6.809,148.699
C00736=1170.938,183.230,-58.903,-178.094,6.808,148.699
C00737=1170.943,182.981,-58.879,-178.097,6.805,148.700
C00738=1170.948,182.733,-58.857,-178.100,6.803,148.700
C00739=1170.952,182.484,-58.834,-178.102,6.801,148.700
C00740=1170.956,182.236,-58.811,-178.105,6.799,148.701
C00741=1170.961,181.986,-58.788,-178.108,6.798,148.701
C00742=1170.966,181.737,-58.765,-178.111,6.795,148.701
C00743=1170.970,181.489,-58.742,-178.114,6.793,148.702
C00744=1170.975,181.240,-58.719,-178.116,6.792,148.702
C00745=1170.979,180.991,-58.697,-178.119,6.789,148.702
C00746=1170.984,180.742,-58.674,-178.121,6.788,148.703
C00747=1170.989,180.493,-58.651,-178.124,6.785,148.703
C00748=1170.994,180.244,-58.629,-178.127,6.783,148.703
C00749=1170.998,179.995,-58.605,-178.130,6.782,148.704
C00750=1171.002,179.746,-58.582,-178.132,6.779,148.704
C00751=1171.008,179.497,-58.560,-178.135,6.778,148.704
C00752=1171.012,179.248,-58.537,-178.138,6.775,148.704
C00753=1171.017,178.999,-58.514,-178.141,6.773,148.705
C00754=1171.021,178.750,-58.492,-178.143,6.772,148.705
C00755=1171.026,178.502,-58.469,-178.146,6.770,148.706
C00756=1171.030,178.252,-58.447,-178.148,6.768,148.706
C00757=1171.035,178.003,-58.424,-178.151,6.766,148.706
C00758=1171.040,177.755,-58.401,-178.154,6.763,148.706
C00759=1171.045,177.506,-58.379,-178.157,6.762,148.707
C00760=1171.049,177.257,-58.356,-178.160,6.760,148.707
C00761=1171.054,177.008,-58.334,-178.162,6.758,148.707
C00762=1171.058,176.759,-58.311,-178.165,6.756,148.708
C00763=1171.063,176.510,-58.288,-178.167,6.754,148.708
C00764=1171.067,176.261,-58.265,-178.170,6.752,148.708
C00765=1171.073,176.012,-58.243,-178.173,6.750,148.709
C00766=1171.077,175.763,-58.220,-178.176,6.748,148.709
C00767=1171.082,175.515,-58.199,-178.178,6.746,148.709
C00768=1171.086,175.266,-58.175,-178.181,6.744,148.710
C00769=1171.091,175.016,-58.153,-178.184,6.743,148.710
C00770=1171.096,174.767,-58.131,-178.186,6.741,148.710
C00771=1171.100,174.519,-58.108,-178.189,6.738,148.711
C00772=1171.104,174.269,-58.086,-178.192,6.736,148.711
C00773=1171.110,174.021,-58.063,-178.195,6.735,148.711
C00774=1171.114,173.772,-58.041,-178.197,6.733,148.712
C00775=1171.119,173.522,-58.018,-178.200,6.731,148.712
C00776=1171.124,173.274,-57.996,-178.203,6.729,148.712
C00777=1171.128,173.025,-57.974,-178.205,6.727,148.713
C00778=1171.133,172.776,-57.951,-178.208,6.725,148.713
C00779=1171.137,172.527,-57.929,-178.211,6.723,148.713
C00780=1171.142,172.277,-57.907,-178.213,6.721,148.714
C00781=1171.147,172.029,-57.885,-178.216,6.719,148.714
C00782=1171.151,171.780,-57.862,-178.219,6.717,148.714
C00783=1171.156,171.531,-57.840,-178.222,6.716,148.715
C00784=1171.161,171.282,-57.818,-178.224,6.714,148.715
C00785=1171.166,171.034,-57.795,-178.227,6.711,148.715
C00786=1171.170,170.784,-57.773,-178.230,6.710,148.716
C00787=1171.174,170.535,-57.751,-178.232,6.708,148.716
C00788=1171.180,170.286,-57.729,-178.235,6.706,148.716
C00789=1171.184,170.037,-57.706,-178.238,6.704,148.717
C00790=1171.189,169.789,-57.684,-178.240,6.702,148.717
C00791=1171.193,169.539,-57.662,-178.243,6.700,148.717
C00792=1171.199,169.290,-57.640,-178.246,6.699,148.718
C00793=1171.203,169.041,-57.618,-178.248,6.697,148.718
C00794=1171.208,168.792,-57.596,-178.252,6.694,148.719
C00795=1171.212,168.544,-57.574,-178.254,6.693,148.719
C00796=1171.217,168.295,-57.552,-178.257,6.691,148.719
C00797=1171.222,168.045,-57.529,-178.260,6.689,148.720
C00798=1171.226,167.797,-57.508,-178.262,6.687,148.720
C00799=1171.231,167.547,-57.485,-178.265,6.685,148.720
C00800=1171.236,167.299,-57.464,-178.267,6.683,148.721
C00801=1171.240,167.049,-57.442,-178.270,6.682,148.721
C00802=1171.245,166.800,-57.419,-178.273,6.680,148.721
C00803=1171.250,166.551,-57.397,-178.275,6.678,148.722
C00804=1171.255,166.302,-57.376,-178.278,6.676,148.722
C00805=1171.259,166.053,-57.354,-178.281,6.674,148.722
C00806=1171.264,165.804,-57.332,-178.284,6.672,148.723
C00807=1171.268,165.555,-57.310,-178.287,6.670,148.723
C00808=1171.273,165.306,-57.288,-178.289,6.669,148.723
C00809=1171.277,165.057,-57.266,-178.292,6.667,148.724
C00810=1171.282,164.808,-57.245,-178.295,6.665,148.724
C00811=1171.288,164.559,-57.222,-178.298,6.663,148.725
C00812=1171.292,164.310,-57.200,-178.300,6.661,148.725
C00813=1171.297,164.061,-57.179,-178.302,6.659,148.725
C00814=1171.301,163.812,-57.156,-178.305,6.658,148.725
C00815=1171.306,163.563,-57.135,-178.308,6.656,148.726
C00816=1171.310,163.314,-57.113,-178.310,6.654,148.726
C00817=1171.315,163.066,-57.091,-178.313,6.652,148.727
C00818=1171.320,162.817,-57.069,-178.316,6.650,148.727
C00819=1171.324,162.568,-57.047,-178.319,6.648,148.727
C00820=1171.329,162.319,-57.026,-178.322,6.646,148.728
C00821=1171.334,162.069,-57.004,-178.324,6.645,148.728
C00822=1171.338,161.820,-56.983,-178.327,6.643,148.728
C00823=1171.343,161.572,-56.961,-178.330,6.641,148.729
C00824=1171.348,161.322,-56.939,-178.333,6.639,148.729
C00825=1171.352,161.074,-56.917,-178.335,6.638,148.730
C00826=1171.357,160.824,-56.895,-178.338,6.636,148.730
C00827=1171.362,160.575,-56.874,-178.341,6.634,148.730
C00828=1171.367,160.326,-56.853,-178.343,6.632,148.731
C00829=1171.371,160.077,-56.830,-178.346,6.630,148.731
C00830=1171.376,159.828,-56.809,-178.349,6.629,148.731
C00831=1171.381,159.579,-56.788,-178.351,6.627,148.732
C00832=1171.385,159.330,-56.766,-178.354,6.625,148.732
C00833=1171.389,159.082,-56.745,-178.357,6.623,148.733
C00834=1171.394,158.833,-56.723,-178.359,6.622,148.733
C00835=1171.400,158.564,-56.700,-178.363,6.619,148.733
C00836=1171.405,158.294,-56.677,-178.365,6.617,148.734
C00837=1171.410,158.025,-56.654,-178.368,6.616,148.734
C00838=1171.415,157.757,-56.630,-178.371,6.614,148.734
C00839=1171.420,157.507,-56.609,-178.373,6.612,148.735
C00840=1171.424,157.258,-56.587,-178.376,6.610,148.735
C00841=1171.429,157.009,-56.565,-178.379,6.609,148.736
C00842=1171.434,156.760,-56.544,-178.382,6.606,148.736
C00843=1171.438,156.511,-56.522,-178.385,6.604,148.736
C00844=1171.443,156.262,-56.501,-178.388,6.603,148.737
C00845=1171.448,156.013,-56.480,-178.390,6.601,148.737
C00846=1171.452,155.765,-56.459,-178.393,6.599,148.737
C00847=1171.457,155.515,-56.437,-178.396,6.597,148.738
C00848=1171.462,155.266,-56.416,-178.398,6.596,148.738
C00849=1171.467,155.017,-56.395,-178.401,6.594,148.739
C00850=1171.471,154.768,-56.374,-178.404,6.592,148.739
C00851=1171.476,154.518,-56.352,-178.406,6.590,148.739
C00852=1171.481,154.270,-56.331,-178.409,6.589,148.740
C00853=1171.486,154.021,-56.310,-178.412,6.587,148.740
C00854=1171.490,153.772,-56.288,-178.414,6.585,148.740
C00855=1171.495,153.522,-56.267,-178.417,6.583,148.741
C00856=1171.499,153.274,-56.245,-178.420,6.582,148.741
C00857=1171.505,153.024,-56.224,-178.423,6.580,148.742
C00858=1171.509,152.776,-56.203,-178.425,6.578,148.742
C00859=1171.514,152.527,-56.182,-178.428,6.576,148.742
C00860=1171.518,152.277,-56.161,-178.431,6.575,148.743
C00861=1171.523,152.028,-56.139,-178.433,6.573,148.743
C00862=1171.528,151.779,-56.119,-178.436,6.571,148.744
C00863=1171.533,151.531,-56.097,-178.439,6.570,148.744
C00864=1171.538,151.281,-56.076,-178.442,6.568,148.744
C00865=1171.542,151.032,-56.056,-178.444,6.567,148.745
C00866=1171.546,150.783,-56.034,-178.447,6.565,148.745
C00867=1171.552,150.534,-56.013,-178.449,6.563,148.746
C00868=1171.556,150.285,-55.993,-178.452,6.562,148.746
C00869=1171.561,150.036,-55.971,-178.455,6.560,148.746
C00870=1171.566,149.787,-55.950,-178.457,6.558,148.747
C00871=1171.570,149.537,-55.929,-178.460,6.556,148.747
C00872=1171.575,149.288,-55.908,-178.463,6.555,148.747
C00873=1171.580,149.039,-55.887,-178.466,6.553,148.748
C00874=1171.584,148.790,-55.866,-178.468,6.551,148.748
C00875=1171.590,148.541,-55.845,-178.471,6.549,148.749
C00876=1171.594,148.293,-55.824,-178.474,6.548,148.749
C00877=1171.599,148.044,-55.803,-178.476,6.546,148.749
C00878=1171.604,147.794,-55.782,-178.479,6.544,148.750
C00879=1171.608,147.545,-55.761,-178.482,6.542,148.750
C00880=1171.613,147.295,-55.741,-178.484,6.541,148.751
C00881=1171.617,147.047,-55.719,-178.487,6.539,148.751
C00882=1171.622,146.798,-55.698,-178.490,6.538,148.752
C00883=1171.627,146.549,-55.678,-178.493,6.536,148.752
C00884=1171.632,146.300,-55.657,-178.496,6.534,148.752
C00885=1171.636,146.051,-55.637,-178.498,6.532,148.753
C00886=1171.642,145.801,-55.616,-178.501,6.531,148.753
C00887=1171.646,145.552,-55.595,-178.504,6.529,148.753
C00888=1171.651,145.304,-55.574,-178.506,6.527,148.754
C00889=1171.655,145.054,-55.553,-178.509,6.526,148.754
C00890=1171.660,144.805,-55.532,-178.511,6.524,148.755
C00891=1171.664,144.556,-55.512,-178.514,6.523,148.755
C00892=1171.670,144.307,-55.491,-178.517,6.521,148.755
C00893=1171.674,144.058,-55.470,-178.519,6.519,148.756
C00894=1171.679,143.808,-55.449,-178.522,6.517,148.756
C00895=1171.684,143.560,-55.429,-178.525,6.516,148.757
C00896=1171.689,143.310,-55.408,-178.528,6.514,148.757
C00897=1171.693,143.061,-55.388,-178.531,6.513,148.758
C00898=1171.698,142.812,-55.367,-178.533,6.511,148.758
C00899=1171.703,142.563,-55.346,-178.536,6.509,148.758
C00900=1171.707,142.314,-55.326,-178.539,6.507,148.759
C00901=1171.712,142.065,-55.305,-178.541,6.506,148.759
C00902=1171.717,141.816,-55.285,-178.544,6.504,148.759
C00903=1171.722,141.567,-55.264,-178.546,6.503,148.760
C00904=1171.727,141.318,-55.243,-178.549,6.501,148.760
C00905=1171.731,141.069,-55.223,-178.552,6.499,148.761
C00906=1171.736,140.820,-55.202,-178.555,6.498,148.761
C00907=1171.741,140.571,-55.182,-178.558,6.496,148.762
C00908=1171.745,140.321,-55.162,-178.560,6.495,148.762
C00909=1171.750,140.072,-55.141,-178.563,6.493,148.762
C00910=1171.755,139.823,-55.121,-178.566,6.491,148.763
C00911=1171.760,139.574,-55.100,-178.568,6.489,148.763
C00912=1171.765,139.325,-55.079,-178.571,6.488,148.764
C00913=1171.769,139.076,-55.059,-178.573,6.487,148.764
C00914=1171.773,138.827,-55.038,-178.576,6.485,148.764
C00915=1171.779,138.577,-55.018,-178.579,6.484,148.765
C00916=1171.783,138.328,-54.998,-178.582,6.482,148.765
C00917=1171.788,138.079,-54.977,-178.584,6.480,148.766
C00918=1171.793,137.830,-54.957,-178.587,6.478,148.766
C00919=1171.797,137.581,-54.936,-178.590,6.477,148.766
C00920=1171.803,137.332,-54.917,-178.593,6.475,148.767
C00921=1171.807,137.083,-54.896,-178.595,6.473,148.767
C00922=1171.812,136.834,-54.876,-178.597,6.472,148.768
C00923=1171.817,136.585,-54.855,-178.601,6.471,148.768
C00924=1171.822,136.335,-54.835,-178.603,6.469,148.769
C00925=1171.826,136.086,-54.815,-178.606,6.467,148.769
C00926=1171.831,135.837,-54.794,-178.609,6.466,148.769
C00927=1171.836,135.587,-54.774,-178.611,6.464,148.770
C00928=1171.840,135.338,-54.754,-178.614,6.462,148.770
C00929=1171.845,135.089,-54.734,-178.617,6.460,148.771
C00930=1171.851,134.840,-54.714,-178.619,6.460,148.771
C00931=1171.855,134.591,-54.693,-178.622,6.458,148.772
C00932=1171.860,134.342,-54.673,-178.625,6.456,148.772
C00933=1171.864,134.093,-54.653,-178.627,6.455,148.772
C00934=1171.869,133.844,-54.633,-178.630,6.453,148.773
C00935=1171.873,133.595,-54.613,-178.633,6.451,148.773
C00936=1171.879,133.345,-54.592,-178.636,6.449,148.774
C00937=1171.884,133.097,-54.572,-178.638,6.449,148.774
C00938=1171.889,132.847,-54.553,-178.641,6.447,148.775
C00939=1171.893,132.579,-54.531,-178.644,6.445,148.775
C00940=1171.899,132.310,-54.509,-178.646,6.444,148.775
C00941=1171.904,132.042,-54.488,-178.650,6.441,148.776
C00942=1171.909,131.773,-54.466,-178.653,6.440,148.776
C00943=1171.914,131.524,-54.446,-178.655,6.439,148.777
C00944=1171.918,131.275,-54.426,-178.658,6.437,148.777
C00945=1171.923,131.025,-54.406,-178.661,6.436,148.778
C00946=1171.927,130.776,-54.386,-178.663,6.434,148.778
C00947=1171.933,130.527,-54.366,-178.666,6.432,148.779
C00948=1171.937,130.278,-54.346,-178.669,6.430,148.779
C00949=1171.942,130.029,-54.326,-178.671,6.429,148.779
C00950=1171.947,129.779,-54.307,-178.674,6.428,148.780
C00951=1171.952,129.531,-54.287,-178.677,6.426,148.780
C00952=1171.957,129.281,-54.267,-178.680,6.425,148.781
C00953=1171.962,129.032,-54.246,-178.682,6.423,148.781
C00954=1171.966,128.783,-54.227,-178.685,6.421,148.782
C00955=1171.972,128.534,-54.207,-178.687,6.420,148.782
C00956=1171.976,128.285,-54.187,-178.690,6.419,148.783
C00957=1171.981,128.035,-54.167,-178.693,6.417,148.783
C00958=1171.985,127.786,-54.147,-178.696,6.415,148.783
C00959=1171.991,127.537,-54.128,-178.698,6.414,148.784
C00960=1171.995,127.288,-54.108,-178.701,6.413,148.784
C00961=1171.999,127.039,-54.088,-178.703,6.411,148.785
C00962=1172.004,126.790,-54.068,-178.706,6.410,148.785
C00963=1172.009,126.541,-54.049,-178.709,6.408,148.786
C00964=1172.014,126.292,-54.029,-178.712,6.406,148.786
C00965=1172.018,126.042,-54.009,-178.715,6.404,148.786
C00966=1172.023,125.793,-53.989,-178.717,6.403,148.787
C00967=1172.029,125.544,-53.970,-178.720,6.402,148.787
C00968=1172.033,125.295,-53.950,-178.723,6.400,148.788
C00969=1172.038,125.045,-53.930,-178.725,6.399,148.788
C00970=1172.043,124.796,-53.911,-178.728,6.397,148.789
C00971=1172.048,124.547,-53.891,-178.730,6.396,148.789
C00972=1172.053,124.297,-53.872,-178.733,6.395,148.790
C00973=1172.058,124.049,-53.852,-178.736,6.393,148.790
C00974=1172.062,123.800,-53.832,-178.739,6.391,148.790
C00975=1172.066,123.550,-53.813,-178.741,6.390,148.791
C00976=1172.072,123.301,-53.794,-178.744,6.389,148.791
C00977=1172.076,123.052,-53.774,-178.747,6.387,148.792
C00978=1172.081,122.803,-53.754,-178.749,6.385,148.792
C00979=1172.086,122.554,-53.734,-178.752,6.384,148.793
C00980=1172.090,122.305,-53.715,-178.754,6.383,148.793
C00981=1172.095,122.055,-53.696,-178.757,6.381,148.794
C00982=1172.100,121.806,-53.676,-178.760,6.380,148.794
C00983=1172.105,121.557,-53.657,-178.763,6.378,148.794
C00984=1172.110,121.307,-53.637,-178.765,6.377,148.795
C00985=1172.115,121.058,-53.618,-178.768,6.375,148.795
C00986=1172.119,120.809,-53.599,-178.771,6.374,148.796
C00987=1172.124,120.560,-53.579,-178.774,6.372,148.796
C00988=1172.129,120.311,-53.560,-178.776,6.370,148.797
C00989=1172.134,120.061,-53.540,-178.778,6.369,148.797
C00990=1172.139,119.812,-53.521,-178.782,6.368,148.798
C00991=1172.143,119.563,-53.502,-178.784,6.366,148.798
C00992=1172.149,119.314,-53.482,-178.787,6.365,148.799
C00993=1172.153,119.064,-53.463,-178.789,6.364,148.799
C00994=1172.157,118.815,-53.444,-178.792,6.362,148.800
C00995=1172.163,118.566,-53.424,-178.795,6.361,148.800
C00996=1172.167,118.317,-53.405,-178.798,6.359,148.800
C00997=1172.173,118.068,-53.385,-178.800,6.358,148.801
C00998=1172.177,117.819,-53.366,-178.803,6.357,148.801
C00999=1172.182,117.570,-53.347,-178.806,6.355,148.802
C01000=1172.187,117.320,-53.327,-178.809,6.353,148.802
C01001=1172.191,117.071,-53.308,-178.811,6.352,148.803
C01002=1172.196,116.822,-53.289,-178.814,6.351,148.803
C01003=1172.201,116.573,-53.269,-178.817,6.349,148.804
C01004=1172.206,116.324,-53.251,-178.819,6.347,148.804
C01005=1172.211,116.074,-53.232,-178.821,6.347,148.804
C01006=1172.216,115.825,-53.212,-178.825,6.345,148.805
C01007=1172.220,115.576,-53.193,-178.827,6.343,148.805
C01008=1172.225,115.327,-53.174,-178.829,6.343,148.806
C01009=1172.230,115.077,-53.154,-178.832,6.341,148.806
C01010=1172.235,114.829,-53.136,-178.835,6.339,148.807
C01011=1172.240,114.578,-53.117,-178.838,6.338,148.807
C01012=1172.245,114.330,-53.097,-178.840,6.337,148.808
C01013=1172.249,114.080,-53.078,-178.843,6.335,148.808
C01014=1172.254,113.831,-53.059,-178.846,6.334,148.809
C01015=1172.259,113.582,-53.041,-178.849,6.332,148.809
C01016=1172.264,113.333,-53.021,-178.851,6.331,148.810
C01017=1172.268,113.083,-53.002,-178.854,6.330,148.810
C01018=1172.273,112.835,-52.983,-178.857,6.328,148.811
C01019=1172.278,112.584,-52.964,-178.859,6.327,148.811
C01020=1172.283,112.336,-52.945,-178.862,6.325,148.811
C01021=1172.288,112.087,-52.926,-178.865,6.324,148.812
C01022=1172.292,111.838,-52.907,-178.868,6.322,148.812
C01023=1172.298,111.588,-52.889,-178.870,6.321,148.813
C01024=1172.302,111.339,-52.870,-178.872,6.320,148.813
C01025=1172.308,111.089,-52.851,-178.876,6.318,148.814
C01026=1172.312,110.840,-52.832,-178.878,6.317,148.814
C01027=1172.317,110.591,-52.813,-178.880,6.316,148.815
C01028=1172.322,110.342,-52.795,-178.884,6.314,148.815
C01029=1172.327,110.093,-52.775,-178.886,6.313,148.816
C01030=1172.331,109.844,-52.756,-178.888,6.312,148.816
C01031=1172.336,109.594,-52.737,-178.891,6.310,148.817
C01032=1172.341,109.345,-52.719,-178.894,6.309,148.817
C01033=1172.346,109.095,-52.700,-178.897,6.308,148.818
C01034=1172.351,108.847,-52.681,-178.899,6.306,148.818
C01035=1172.356,108.598,-52.662,-178.902,6.305,148.819
C01036=1172.360,108.348,-52.643,-178.905,6.304,148.819
C01037=1172.365,108.099,-52.625,-178.907,6.302,148.820
C01038=1172.371,107.850,-52.606,-178.910,6.301,148.820
C01039=1172.375,107.601,-52.587,-178.913,6.300,148.821
C01040=1172.380,107.351,-52.568,-178.915,6.298,148.821
C01041=1172.384,107.102,-52.549,-178.918,6.296,148.821
C01042=1172.390,106.852,-52.531,-178.921,6.296,148.822
C01043=1172.395,106.584,-52.511,-178.923,6.294,148.822
C01044=1172.400,106.315,-52.490,-178.927,6.293,148.823
C01045=1172.405,106.047,-52.471,-178.929,6.291,148.823
C01046=1172.410,105.779,-52.450,-178.932,6.289,148.824
C01047=1172.415,105.530,-52.432,-178.935,6.289,148.825
C01048=1172.420,105.280,-52.414,-178.937,6.287,148.825
C01049=1172.425,105.031,-52.395,-178.941,6.286,148.826
C01050=1172.430,104.782,-52.377,-178.943,6.285,148.826
C01051=1172.434,104.533,-52.358,-178.945,6.283,148.826
C01052=1172.440,104.283,-52.339,-178.949,6.282,148.827
C01053=1172.445,104.034,-52.321,-178.951,6.281,148.827
C01054=1172.449,103.785,-52.302,-178.953,6.279,148.828
C01055=1172.454,103.535,-52.283,-178.957,6.278,148.828
C01056=1172.459,103.286,-52.265,-178.959,6.277,148.829
C01057=1172.463,103.037,-52.246,-178.961,6.275,148.829
C01058=1172.469,102.788,-52.228,-178.965,6.274,148.830
C01059=1172.474,102.538,-52.210,-178.967,6.273,148.830
C01060=1172.478,102.290,-52.191,-178.970,6.271,148.831
C01061=1172.483,102.040,-52.173,-178.973,6.270,148.831
C01062=1172.488,101.790,-52.154,-178.975,6.269,148.832
C01063=1172.493,101.541,-52.136,-178.978,6.267,148.832
C01064=1172.498,101.293,-52.117,-178.981,6.266,148.833
C01065=1172.502,101.043,-52.099,-178.983,6.265,148.833
C01066=1172.508,100.793,-52.081,-178.986,6.263,148.834
C01067=1172.513,100.544,-52.063,-178.988,6.262,148.834
C01068=1172.517,100.296,-52.044,-178.991,6.261,148.835
C01069=1172.522,100.046,-52.025,-178.994,6.259,148.835
C01070=1172.526,99.797,-52.008,-178.996,6.258,148.836
C01071=1172.532,99.547,-51.989,-178.999,6.257,148.836
C01072=1172.537,99.298,-51.971,-179.002,6.255,148.837
C01073=1172.541,99.049,-51.952,-179.004,6.254,148.837
C01074=1172.546,98.799,-51.934,-179.007,6.253,148.838
C01075=1172.551,98.550,-51.916,-179.009,6.252,148.838
C01076=1172.556,98.301,-51.898,-179.012,6.251,148.839
C01077=1172.561,98.052,-51.879,-179.015,6.249,148.839
C01078=1172.566,97.802,-51.861,-179.017,6.248,148.840
C01079=1172.571,97.553,-51.843,-179.020,6.247,148.840
C01080=1172.576,97.303,-51.825,-179.023,6.246,148.841
C01081=1172.580,97.054,-51.807,-179.026,6.244,148.841
C01082=1172.585,96.806,-51.788,-179.029,6.243,148.842
C01083=1172.589,96.556,-51.770,-179.031,6.242,148.842
C01084=1172.594,96.307,-51.752,-179.034,6.240,148.843
C01085=1172.600,96.057,-51.734,-179.036,6.239,148.843
C01086=1172.605,95.808,-51.716,-179.039,6.238,148.844
C01087=1172.610,95.559,-51.698,-179.042,6.236,148.844
C01088=1172.615,95.310,-51.680,-179.044,6.235,148.845
C01089=1172.620,95.060,-51.662,-179.047,6.234,148.845
C01090=1172.624,94.811,-51.643,-179.049,6.233,148.846
C01091=1172.629,94.561,-51.625,-179.052,6.232,148.846
C01092=1172.634,94.312,-51.607,-179.055,6.230,148.847
C01093=1172.639,94.063,-51.589,-179.057,6.229,148.847
C01094=1172.644,93.814,-51.571,-179.060,6.228,148.848
C01095=1172.648,93.565,-51.553,-179.063,6.227,148.848
C01096=1172.653,93.315,-51.535,-179.066,6.225,148.849
C01097=1172.658,93.065,-51.518,-179.068,6.224,148.849
C01098=1172.663,92.816,-51.500,-179.071,6.223,148.850
C01099=1172.668,92.567,-51.482,-179.074,6.221,148.850
C01100=1172.673,92.317,-51.464,-179.076,6.221,148.851
C01101=1172.678,92.068,-51.446,-179.079,6.219,148.851
C01102=1172.683,91.819,-51.428,-179.081,6.218,148.852
C01103=1172.687,91.570,-51.410,-179.084,6.217,148.852
C01104=1172.692,91.321,-51.392,-179.087,6.215,148.853
C01105=1172.697,91.072,-51.374,-179.089,6.214,148.853
C01106=1172.703,90.822,-51.357,-179.092,6.213,148.854
C01107=1172.707,90.573,-51.339,-179.094,6.212,148.854
C01108=1172.712,90.323,-51.321,-179.098,6.211,148.855
C01109=1172.717,90.074,-51.302,-179.100,6.210,148.855
C01110=1172.722,89.824,-51.284,-179.103,6.208,148.856
C01111=1172.727,89.575,-51.267,-179.106,6.207,148.856
C01112=1172.732,89.325,-51.249,-179.108,6.206,148.857
C01113=1172.736,89.077,-51.232,-179.111,6.204,148.857
C01114=1172.741,88.827,-51.214,-179.113,6.204,148.858
C01115=1172.746,88.578,-51.196,-179.116,6.202,148.858
C01116=1172.751,88.328,-51.178,-179.119,6.201,148.859
C01117=1172.756,88.079,-51.161,-179.121,6.200,148.859
C01118=1172.761,87.830,-51.143,-179.124,6.199,148.860
C01119=1172.766,87.580,-51.125,-179.127,6.197,148.860
C01120=1172.771,87.331,-51.107,-179.129,6.196,148.861
C01121=1172.775,87.082,-51.090,-179.132,6.195,148.861
C01122=1172.780,86.832,-51.073,-179.135,6.193,148.862
C01123=1172.785,86.583,-51.055,-179.137,6.193,148.863
C01124=1172.790,86.334,-51.037,-179.140,6.191,148.863
C01125=1172.795,86.084,-51.019,-179.142,6.190,148.863
C01126=1172.800,85.835,-51.001,-179.145,6.189,148.864
C01127=1172.804,85.586,-50.984,-179.148,6.188,148.864
C01128=1172.810,85.336,-50.967,-179.151,6.187,148.865
C01129=1172.814,85.087,-50.949,-179.153,6.186,148.866
C01130=1172.820,84.837,-50.932,-179.156,6.184,148.866
C01131=1172.825,84.588,-50.914,-179.158,6.184,148.867
C01132=1172.829,84.339,-50.896,-179.161,6.182,148.867
C01133=1172.834,84.090,-50.879,-179.164,6.181,148.868
C01134=1172.839,83.840,-50.861,-179.166,6.180,148.868
C01135=1172.844,83.591,-50.844,-179.169,6.179,148.869
C01136=1172.849,83.343,-50.827,-179.172,6.177,148.869
C01137=1172.854,83.093,-50.809,-179.174,6.177,148.870
C01138=1172.859,82.844,-50.791,-179.177,6.175,148.870
C01139=1172.864,82.594,-50.774,-179.179,6.174,148.871
C01140=1172.868,82.345,-50.757,-179.182,6.173,148.871
C01141=1172.874,82.095,-50.739,-179.185,6.172,148.872
C01142=1172.879,81.846,-50.722,-179.188,6.171,148.872
C01143=1172.883,81.596,-50.705,-179.190,6.170,148.873
C01144=1172.888,81.347,-50.687,-179.193,6.168,148.873
C01145=1172.893,81.097,-50.670,-179.196,6.167,148.874
C01146=1172.898,80.848,-50.652,-179.198,6.166,148.874
C01147=1172.903,80.580,-50.634,-179.201,6.165,148.875
C01148=1172.909,80.312,-50.615,-179.204,6.164,148.876
C01149=1172.914,80.043,-50.596,-179.207,6.162,148.876
C01150=1172.919,79.775,-50.578,-179.210,6.161,148.877
C01151=1172.924,79.526,-50.561,-179.212,6.160,148.877
C01152=1172.929,79.276,-50.543,-179.215,6.159,148.878
C01153=1172.934,79.027,-50.526,-179.217,6.158,148.878
C01154=1172.939,78.777,-50.509,-179.220,6.157,148.879
C01155=1172.944,78.528,-50.491,-179.223,6.156,148.879
C01156=1172.948,78.279,-50.474,-179.225,6.154,148.880
C01157=1172.954,78.029,-50.457,-179.228,6.153,148.880
C01158=1172.958,77.781,-50.440,-179.231,6.152,148.881
C01159=1172.964,77.531,-50.423,-179.233,6.151,148.881
C01160=1172.969,77.281,-50.405,-179.236,6.149,148.882
C01161=1172.973,77.032,-50.388,-179.239,6.149,148.883
C01162=1172.978,76.782,-50.371,-179.241,6.147,148.883
C01163=1172.983,76.534,-50.354,-179.244,6.147,148.884
C01164=1172.988,76.284,-50.336,-179.246,6.146,148.884
C01165=1172.993,76.035,-50.320,-179.249,6.145,148.885
C01166=1172.998,75.785,-50.303,-179.252,6.144,148.885
C01167=1173.003,75.535,-50.285,-179.254,6.142,148.886
C01168=1173.007,75.286,-50.268,-179.257,6.141,148.886
C01169=1173.013,75.037,-50.251,-179.260,6.140,148.887
C01170=1173.017,74.788,-50.234,-179.262,6.139,148.887
C01171=1173.023,74.538,-50.217,-179.265,6.137,148.888
C01172=1173.027,74.289,-50.200,-179.268,6.137,148.888
C01173=1173.033,74.040,-50.183,-179.270,6.135,148.889
C01174=1173.037,73.791,-50.166,-179.273,6.135,148.889
C01175=1173.042,73.541,-50.149,-179.276,6.133,148.890
C01176=1173.047,73.291,-50.132,-179.278,6.133,148.891
C01177=1173.052,73.042,-50.115,-179.280,6.132,148.891
C01178=1173.057,72.793,-50.099,-179.284,6.130,148.892
C01179=1173.062,72.543,-50.082,-179.286,6.129,148.892
C01180=1173.067,72.294,-50.064,-179.289,6.128,148.892
C01181=1173.071,72.045,-50.047,-179.291,6.127,148.893
C01182=1173.077,71.796,-50.030,-179.294,6.126,148.894
C01183=1173.081,71.546,-50.014,-179.297,6.125,148.894
C01184=1173.087,71.296,-49.996,-179.299,6.123,148.895
C01185=1173.092,71.047,-49.980,-179.302,6.123,148.895
C01186=1173.097,70.798,-49.963,-179.304,6.122,148.896
C01187=1173.101,70.548,-49.946,-179.307,6.121,148.896
C01188=1173.106,70.299,-49.930,-179.309,6.120,148.897
C01189=1173.112,70.050,-49.913,-179.313,6.118,148.897
C01190=1173.116,69.800,-49.896,-179.315,6.117,148.898
C01191=1173.121,69.551,-49.879,-179.318,6.116,148.899
C01192=1173.126,69.302,-49.862,-179.320,6.115,148.899
C01193=1173.131,69.052,-49.846,-179.323,6.115,148.900
C01194=1173.136,68.802,-49.828,-179.325,6.113,148.900
C01195=1173.141,68.553,-49.812,-179.328,6.113,148.901
C01196=1173.146,68.304,-49.796,-179.331,6.111,148.901
C01197=1173.151,68.054,-49.778,-179.333,6.110,148.902
C01198=1173.155,67.805,-49.762,-179.336,6.109,148.902
C01199=1173.160,67.556,-49.745,-179.339,6.108,148.903
C01200=1173.166,67.306,-49.728,-179.341,6.107,148.903
C01201=1173.170,67.057,-49.711,-179.344,6.106,148.904
C01202=1173.175,66.808,-49.695,-179.346,6.105,148.904
C01203=1173.180,66.558,-49.678,-179.350,6.104,148.905
C01204=1173.186,66.309,-49.662,-179.352,6.103,148.906
C01205=1173.190,66.059,-49.646,-179.354,6.102,148.906
C01206=1173.195,65.810,-49.629,-179.357,6.101,148.907
C01207=1173.201,65.561,-49.612,-179.359,6.100,148.907
C01208=1173.205,65.311,-49.595,-179.362,6.098,148.908
C01209=1173.210,65.062,-49.579,-179.365,6.098,148.908
C01210=1173.215,64.813,-49.562,-179.367,6.097,148.909
C01211=1173.220,64.562,-49.546,-179.370,6.095,148.909
C01212=1173.225,64.314,-49.529,-179.373,6.095,148.910
C01213=1173.230,64.064,-49.513,-179.375,6.093,148.910
C01214=1173.234,63.815,-49.496,-179.378,6.093,148.911
C01215=1173.239,63.566,-49.480,-179.380,6.092,148.911
C01216=1173.245,63.315,-49.463,-179.383,6.090,148.912
C01217=1173.250,63.067,-49.447,-179.385,6.089,148.913
C01218=1173.254,62.817,-49.430,-179.389,6.088,148.913
C01219=1173.259,62.568,-49.414,-179.391,6.088,148.914
C01220=1173.264,62.318,-49.398,-179.393,6.087,148.914
C01221=1173.269,62.069,-49.381,-179.397,6.085,148.915
C01222=1173.275,61.820,-49.364,-179.399,6.085,148.915
C01223=1173.279,61.570,-49.349,-179.401,6.084,148.916
C01224=1173.284,61.321,-49.332,-179.404,6.082,148.917
C01225=1173.289,61.071,-49.316,-179.407,6.082,148.917
C01226=1173.293,60.822,-49.299,-179.410,6.080,148.918
C01227=1173.300,60.572,-49.283,-179.412,6.080,148.918
C01228=1173.304,60.323,-49.266,-179.414,6.079,148.919
C01229=1173.309,60.073,-49.250,-179.418,6.077,148.919
C01230=1173.314,59.824,-49.234,-179.420,6.077,148.920
C01231=1173.319,59.575,-49.217,-179.422,6.076,148.920
C01232=1173.324,59.325,-49.202,-179.425,6.074,148.921
C01233=1173.329,59.076,-49.185,-179.428,6.074,148.922
C01234=1173.333,58.827,-49.169,-179.430,6.073,148.922
C01235=1173.339,58.577,-49.152,-179.433,6.072,148.923
C01236=1173.344,58.327,-49.136,-179.435,6.071,148.923
C01237=1173.349,58.078,-49.120,-179.439,6.069,148.924
C01238=1173.354,57.829,-49.103,-179.441,6.069,148.924
C01239=1173.359,57.579,-49.088,-179.443,6.068,148.925
C01240=1173.364,57.330,-49.071,-179.446,6.066,148.925
C01241=1173.369,57.081,-49.055,-179.449,6.066,148.926
C01242=1173.373,56.831,-49.039,-179.451,6.065,148.926
C01243=1173.379,56.582,-49.023,-179.454,6.064,148.927
C01244=1173.383,56.332,-49.007,-179.456,6.063,148.928
C01245=1173.388,56.083,-48.990,-179.459,6.062,148.928
C01246=1173.393,55.833,-48.974,-179.462,6.061,148.929
C01247=1173.398,55.584,-48.958,-179.464,6.060,148.929
C01248=1173.403,55.334,-48.942,-179.467,6.060,148.930
C01249=1173.408,55.085,-48.926,-179.470,6.058,148.930
C01250=1173.414,54.836,-48.910,-179.472,6.057,148.931
C01251=1173.419,54.567,-48.893,-179.475,6.056,148.931
C01252=1173.424,54.298,-48.876,-179.478,6.055,148.932
C01253=1173.429,54.030,-48.858,-179.481,6.054,148.933
C01254=1173.434,53.761,-48.841,-179.483,6.053,148.933
C01255=1173.440,53.512,-48.825,-179.486,6.053,148.934
C01256=1173.445,53.263,-48.809,-179.489,6.051,148.935
C01257=1173.450,53.013,-48.793,-179.491,6.050,148.935
C01258=1173.455,52.764,-48.777,-179.494,6.050,148.936
C01259=1173.459,52.514,-48.761,-179.496,6.048,148.936
C01260=1173.465,52.265,-48.745,-179.499,6.048,148.937
C01261=1173.470,52.015,-48.729,-179.501,6.047,148.937
C01262=1173.475,51.766,-48.713,-179.504,6.046,148.938
C01263=1173.480,51.516,-48.697,-179.507,6.045,148.938
C01264=1173.485,51.266,-48.681,-179.509,6.044,148.939
C01265=1173.490,51.017,-48.665,-179.512,6.043,148.940
C01266=1173.495,50.768,-48.650,-179.515,6.042,148.940
C01267=1173.499,50.518,-48.634,-179.517,6.041,148.941
C01268=1173.504,50.270,-48.618,-179.519,6.041,148.941
C01269=1173.510,50.020,-48.602,-179.523,6.039,148.942
C01270=1173.515,49.770,-48.586,-179.525,6.038,148.942
C01271=1173.520,49.521,-48.571,-179.527,6.038,148.943
C01272=1173.524,49.271,-48.554,-179.530,6.036,148.943
C01273=1173.529,49.022,-48.539,-179.533,6.036,148.944
C01274=1173.535,48.773,-48.523,-179.535,6.035,148.945
C01275=1173.539,48.523,-48.507,-179.538,6.034,148.945
C01276=1173.544,48.274,-48.491,-179.541,6.033,148.946
C01277=1173.550,48.024,-48.475,-179.543,6.032,148.946
C01278=1173.555,47.774,-48.460,-179.546,6.032,148.947
C01279=1173.559,47.525,-48.445,-179.548,6.030,148.947
C01280=1173.565,47.276,-48.429,-179.551,6.029,148.948
C01281=1173.569,47.026,-48.413,-179.553,6.029,148.949
C01282=1173.574,46.777,-48.397,-179.556,6.027,148.949
C01283=1173.580,46.527,-48.381,-179.558,6.026,148.950
C01284=1173.584,46.278,-48.366,-179.561,6.026,148.950
C01285=1173.589,46.028,-48.350,-179.564,6.025,148.951
C01286=1173.595,45.779,-48.335,-179.566,6.024,148.951
C01287=1173.600,45.529,-48.319,-179.569,6.023,148.952
C01288=1173.604,45.280,-48.304,-179.571,6.022,148.953
C01289=1173.609,45.031,-48.287,-179.574,6.021,148.953
C01290=1173.615,44.781,-48.272,-179.577,6.020,148.954
C01291=1173.619,44.531,-48.256,-179.579,6.020,148.954
C01292=1173.624,44.282,-48.241,-179.582,6.019,148.955
C01293=1173.629,44.033,-48.225,-179.585,6.018,148.955
C01294=1173.635,43.783,-48.210,-179.587,6.017,148.956
C01295=1173.639,43.534,-48.194,-179.589,6.016,148.957
C01296=1173.644,43.284,-48.179,-179.592,6.016,148.957
C01297=1173.650,43.035,-48.163,-179.595,6.014,148.958
C01298=1173.654,42.786,-48.148,-179.597,6.013,148.958
C01299=1173.659,42.536,-48.132,-179.600,6.013,148.959
C01300=1173.664,42.286,-48.117,-179.602,6.012,148.960
C01301=1173.669,42.037,-48.102,-179.606,6.011,148.960
C01302=1173.674,41.788,-48.086,-179.608,6.010,148.961
C01303=1173.679,41.538,-48.070,-179.610,6.009,148.961
C01304=1173.684,41.289,-48.055,-179.612,6.009,148.962
C01305=1173.689,41.039,-48.039,-179.616,6.007,148.962
C01306=1173.695,40.790,-48.024,-179.618,6.007,148.963
C01307=1173.699,40.541,-48.009,-179.620,6.006,148.964
C01308=1173.704,40.291,-47.993,-179.623,6.005,148.964
C01309=1173.709,40.041,-47.977,-179.626,6.004,148.965
C01310=1173.714,39.791,-47.963,-179.629,6.003,148.965
C01311=1173.720,39.542,-47.947,-179.631,6.002,148.966
C01312=1173.724,39.293,-47.932,-179.633,6.002,148.966
C01313=1173.730,39.044,-47.917,-179.637,6.001,148.967
C01314=1173.735,38.793,-47.901,-179.639,6.000,148.968
C01315=1173.739,38.544,-47.886,-179.641,5.999,148.968
C01316=1173.745,38.295,-47.870,-179.644,5.998,148.969
C01317=1173.750,38.045,-47.856,-179.647,5.997,148.969
C01318=1173.755,37.796,-47.840,-179.649,5.996,148.970
C01319=1173.760,37.546,-47.825,-179.652,5.996,148.970
C01320=1173.764,37.297,-47.809,-179.654,5.995,148.971
C01321=1173.770,37.047,-47.794,-179.657,5.994,148.972
C01322=1173.774,36.798,-47.779,-179.660,5.993,148.972
C01323=1173.780,36.548,-47.764,-179.662,5.992,148.973
C01324=1173.785,36.299,-47.749,-179.664,5.992,148.973
C01325=1173.790,36.050,-47.733,-179.667,5.991,148.974
C01326=1173.795,35.801,-47.718,-179.670,5.990,148.975
C01327=1173.800,35.550,-47.703,-179.672,5.989,148.975
C01328=1173.805,35.301,-47.688,-179.675,5.988,148.976
C01329=1173.810,35.051,-47.673,-179.677,5.988,148.976
C01330=1173.815,34.802,-47.658,-179.680,5.987,148.977
C01331=1173.820,34.552,-47.643,-179.683,5.986,148.977
C01332=1173.825,34.303,-47.628,-179.685,5.985,148.978
C01333=1173.830,34.054,-47.612,-179.687,5.984,148.979
C01334=1173.835,33.804,-47.598,-179.690,5.984,148.979
C01335=1173.841,33.555,-47.582,-179.693,5.982,148.980
C01336=1173.845,33.305,-47.567,-179.695,5.982,148.980
C01337=1173.850,33.055,-47.553,-179.698,5.981,148.981
C01338=1173.855,32.806,-47.537,-179.700,5.980,148.981
C01339=1173.860,32.557,-47.522,-179.703,5.980,148.982
C01340=1173.865,32.307,-47.507,-179.706,5.978,148.983
C01341=1173.870,32.058,-47.492,-179.708,5.978,148.983
C01342=1173.875,31.808,-47.477,-179.711,5.977,148.984
C01343=1173.880,31.558,-47.462,-179.713,5.976,148.984
C01344=1173.885,31.309,-47.447,-179.716,5.976,148.985
C01345=1173.891,31.059,-47.433,-179.718,5.974,148.986
C01346=1173.895,30.810,-47.418,-179.721,5.974,148.986
C01347=1173.901,30.561,-47.402,-179.724,5.973,148.987
C01348=1173.906,30.311,-47.388,-179.726,5.972,148.987
C01349=1173.910,30.062,-47.373,-179.729,5.972,148.988
C01350=1173.916,29.812,-47.358,-179.731,5.971,148.988
C01351=1173.921,29.563,-47.343,-179.734,5.970,148.989
C01352=1173.926,29.313,-47.329,-179.737,5.969,148.990
C01353=1173.931,29.064,-47.313,-179.739,5.968,148.990
C01354=1173.936,28.814,-47.299,-179.741,5.968,148.991
C01355=1173.941,28.545,-47.283,-179.745,5.966,148.992
C01356=1173.947,28.277,-47.266,-179.747,5.966,148.992
C01357=1173.952,28.008,-47.250,-179.749,5.965,148.993
C01358=1173.958,27.739,-47.234,-179.753,5.964,148.993
C01359=1173.963,27.489,-47.220,-179.755,5.963,148.994
C01360=1173.967,27.240,-47.205,-179.758,5.962,148.995
C01361=1173.973,26.990,-47.190,-179.760,5.962,148.995
C01362=1173.978,26.740,-47.176,-179.763,5.962,148.996
C01363=1173.983,26.491,-47.161,-179.765,5.961,148.996
C01364=1173.988,26.242,-47.146,-179.768,5.959,148.997
C01365=1173.993,25.992,-47.131,-179.770,5.959,148.998
C01366=1173.998,25.742,-47.116,-179.773,5.958,148.998
C01367=1174.003,25.493,-47.101,-179.776,5.958,148.999
C01368=1174.008,25.244,-47.087,-179.778,5.957,148.999
C01369=1174.013,24.994,-47.072,-179.780,5.956,149.000
C01370=1174.018,24.745,-47.057,-179.783,5.955,149.000
C01371=1174.023,24.495,-47.043,-179.786,5.954,149.001
C01372=1174.028,24.245,-47.029,-179.789,5.954,149.002
C01373=1174.033,23.996,-47.013,-179.791,5.953,149.002
C01374=1174.038,23.746,-46.999,-179.793,5.952,149.003
C01375=1174.043,23.496,-46.985,-179.796,5.952,149.004
C01376=1174.048,23.247,-46.970,-179.798,5.951,149.004
C01377=1174.053,22.998,-46.956,-179.801,5.950,149.005
C01378=1174.059,22.748,-46.941,-179.804,5.949,149.005
C01379=1174.064,22.499,-46.926,-179.806,5.948,149.006
C01380=1174.069,22.249,-46.912,-179.809,5.948,149.007
C01381=1174.074,22.000,-46.897,-179.811,5.947,149.007
C01382=1174.078,21.750,-46.883,-179.814,5.946,149.008
C01383=1174.083,21.501,-46.868,-179.816,5.946,149.008
C01384=1174.089,21.251,-46.853,-179.818,5.945,149.009
C01385=1174.094,21.001,-46.839,-179.822,5.944,149.010
C01386=1174.099,20.751,-46.825,-179.824,5.943,149.010
C01387=1174.104,20.503,-46.810,-179.826,5.943,149.011
C01388=1174.109,20.253,-46.796,-179.829,5.942,149.011
C01389=1174.114,20.004,-46.781,-179.831,5.941,149.012
C01390=1174.119,19.754,-46.767,-179.834,5.941,149.012
C01391=1174.124,19.504,-46.753,-179.836,5.940,149.013
C01392=1174.129,19.255,-46.737,-179.839,5.939,149.014
C01393=1174.134,19.005,-46.723,-179.842,5.938,149.014
C01394=1174.140,18.756,-46.709,-179.844,5.937,149.015
C01395=1174.145,18.506,-46.695,-179.847,5.937,149.015
C01396=1174.150,18.257,-46.680,-179.849,5.936,149.016
C01397=1174.155,18.007,-46.666,-179.852,5.935,149.017
C01398=1174.159,17.758,-46.651,-179.854,5.935,149.017
C01399=1174.164,17.508,-46.637,-179.856,5.934,149.018
C01400=1174.170,17.259,-46.623,-179.859,5.934,149.018
C01401=1174.175,17.009,-46.609,-179.862,5.932,149.019
C01402=1174.180,16.760,-46.594,-179.864,5.932,149.020
C01403=1174.185,16.510,-46.580,-179.867,5.931,149.020
C01404=1174.190,16.260,-46.566,-179.870,5.931,149.021
C01405=1174.195,16.011,-46.552,-179.872,5.930,149.021
C01406=1174.200,15.762,-46.538,-179.875,5.929,149.022
C01407=1174.205,15.512,-46.523,-179.877,5.928,149.022
C01408=1174.210,15.262,-46.509,-179.879,5.928,149.023
C01409=1174.215,15.012,-46.495,-179.882,5.927,149.024
C01410=1174.220,14.763,-46.481,-179.884,5.927,149.024
C01411=1174.225,14.514,-46.467,-179.887,5.925,149.025
C01412=1174.230,14.265,-46.452,-179.890,5.925,149.026
C01413=1174.235,14.015,-46.437,-179.892,5.924,149.026
C01414=1174.240,13.765,-46.424,-179.895,5.924,149.027
C01415=1174.246,13.516,-46.410,-179.897,5.923,149.027
C01416=1174.251,13.266,-46.396,-179.900,5.922,149.028
C01417=1174.256,13.016,-46.381,-179.902,5.922,149.029
C01418=1174.261,12.766,-46.367,-179.905,5.921,149.029
C01419=1174.266,12.517,-46.353,-179.907,5.920,149.030
C01420=1174.271,12.268,-46.339,-179.910,5.920,149.030
C01421=1174.276,12.018,-46.325,-179.912,5.919,149.031
C01422=1174.281,11.768,-46.310,-179.915,5.918,149.032
C01423=1174.287,11.519,-46.296,-179.918,5.917,149.032
C01424=1174.292,11.270,-46.282,-179.920,5.916,149.033
C01425=1174.297,11.020,-46.268,-179.923,5.916,149.033
C01426=1174.302,10.770,-46.254,-179.925,5.915,149.034
C01427=1174.306,10.521,-46.240,-179.928,5.915,149.035
C01428=1174.311,10.272,-46.226,-179.930,5.914,149.035
C01429=1174.317,10.021,-46.212,-179.932,5.913,149.036
C01430=1174.322,9.772,-46.199,-179.935,5.913,149.036
C01431=1174.327,9.523,-46.184,-179.938,5.912,149.037
C01432=1174.332,9.273,-46.170,-179.940,5.912,149.038
C01433=1174.337,9.023,-46.156,-179.943,5.911,149.038
C01434=1174.343,8.774,-46.142,-179.945,5.911,149.039
C01435=1174.347,8.524,-46.129,-179.947,5.910,149.039
C01436=1174.352,8.275,-46.115,-179.951,5.909,149.040
C01437=1174.358,8.026,-46.101,-179.953,5.908,149.041
C01438=1174.363,7.776,-46.086,-179.955,5.907,149.041
C01439=1174.368,7.526,-46.072,-179.958,5.907,149.042
C01440=1174.373,7.276,-46.059,-179.960,5.906,149.042
C01441=1174.378,7.027,-46.045,-179.963,5.905,149.043
C01442=1174.383,6.777,-46.031,-179.966,5.905,149.044
C01443=1174.388,6.528,-46.017,-179.968,5.904,149.044
C01444=1174.393,6.278,-46.003,-179.970,5.904,149.045
C01445=1174.398,6.029,-45.990,-179.973,5.903,149.046
C01446=1174.403,5.780,-45.976,-179.975,5.902,149.046
C01447=1174.408,5.530,-45.962,-179.978,5.902,149.047
C01448=1174.413,5.280,-45.948,-179.980,5.901,149.047
C01449=1174.419,5.031,-45.934,-179.983,5.901,149.048
C01450=1174.423,4.781,-45.920,-179.985,5.900,149.049
C01451=1174.429,4.532,-45.907,-179.987,5.899,149.049
C01452=1174.434,4.282,-45.893,-179.990,5.899,149.050
C01453=1174.439,4.032,-45.879,-179.993,5.898,149.050
C01454=1174.444,3.783,-45.866,-179.995,5.897,149.051
C01455=1174.449,3.533,-45.852,-179.998,5.897,149.052
C01456=1174.454,3.283,-45.838,180.000,5.897,149.052
C01457=1174.459,3.034,-45.825,179.998,5.896,149.053
C01458=1174.464,2.784,-45.811,179.995,5.895,149.053
C01459=1174.469,2.515,-45.796,179.992,5.894,149.054
C01460=1174.475,2.246,-45.781,179.989,5.894,149.055
C01461=1174.481,1.977,-45.766,179.986,5.893,149.055
C01462=1174.487,1.707,-45.752,179.984,5.892,149.056
C01463=1174.491,1.458,-45.738,179.982,5.892,149.057
C01464=1174.496,1.208,-45.724,179.979,5.891,149.057
C01465=1174.502,0.958,-45.711,179.977,5.890,149.058
C01466=1174.506,0.709,-45.697,179.974,5.890,149.058
C01467=1174.512,0.459,-45.684,179.971,5.890,149.059
C01468=1174.517,0.210,-45.670,179.969,5.889,149.060
C01469=1174.522,-0.040,-45.657,179.967,5.888,149.060
C01470=1174.527,-0.289,-45.643,179.964,5.888,149.061
C01471=1174.532,-0.539,-45.630,179.962,5.887,149.061
C01472=1174.537,-0.788,-45.616,179.959,5.886,149.062
C01473=1174.543,-1.038,-45.603,179.956,5.886,149.063
C01474=1174.548,-1.287,-45.589,179.954,5.885,149.063
C01475=1174.553,-1.537,-45.576,179.952,5.885,149.064
C01476=1174.558,-1.787,-45.561,179.949,5.884,149.064
C01477=1174.563,-2.036,-45.549,179.947,5.883,149.065
C01478=1174.568,-2.286,-45.534,179.944,5.883,149.066
C01479=1174.573,-2.535,-45.522,179.942,5.882,149.066
C01480=1174.578,-2.785,-45.508,179.939,5.882,149.067
C01481=1174.583,-3.034,-45.495,179.937,5.881,149.068
C01482=1174.588,-3.285,-45.481,179.935,5.880,149.068
C01483=1174.594,-3.534,-45.468,179.932,5.880,149.069
C01484=1174.598,-3.784,-45.455,179.929,5.879,149.069
C01485=1174.604,-4.033,-45.441,179.927,5.879,149.070
C01486=1174.608,-4.283,-45.428,179.924,5.878,149.071
C01487=1174.614,-4.533,-45.415,179.922,5.878,149.071
C01488=1174.619,-4.782,-45.401,179.920,5.877,149.072
C01489=1174.624,-5.032,-45.388,179.917,5.876,149.072
C01490=1174.629,-5.282,-45.375,179.914,5.876,149.073
C01491=1174.634,-5.531,-45.361,179.912,5.875,149.074
C01492=1174.640,-5.780,-45.348,179.909,5.875,149.074
C01493=1174.645,-6.030,-45.335,179.907,5.874,149.075
C01494=1174.650,-6.279,-45.321,179.905,5.873,149.075
C01495=1174.655,-6.529,-45.308,179.902,5.873,149.076
C01496=1174.660,-6.779,-45.295,179.899,5.872,149.077
C01497=1174.665,-7.028,-45.281,179.897,5.872,149.077
C01498=1174.670,-7.278,-45.268,179.894,5.871,149.078
C01499=1174.675,-7.528,-45.255,179.892,5.870,149.078
C01500=1174.680,-7.777,-45.241,179.890,5.870,149.079
C01501=1174.686,-8.026,-45.228,179.887,5.869,149.080
C01502=1174.691,-8.276,-45.215,179.885,5.869,149.080
C01503=1174.696,-8.526,-45.202,179.882,5.868,149.081
C01504=1174.701,-8.775,-45.188,179.879,5.868,149.082
C01505=1174.706,-9.025,-45.176,179.877,5.867,149.082
C01506=1174.711,-9.275,-45.162,179.875,5.866,149.083
C01507=1174.716,-9.524,-45.150,179.872,5.866,149.084
C01508=1174.722,-9.773,-45.136,179.870,5.865,149.084
C01509=1174.726,-10.023,-45.123,179.867,5.865,149.085
C01510=1174.732,-10.273,-45.109,179.864,5.864,149.085
C01511=1174.737,-10.523,-45.097,179.862,5.863,149.086
C01512=1174.742,-10.772,-45.084,179.860,5.863,149.087
C01513=1174.748,-11.022,-45.071,179.857,5.862,149.087
C01514=1174.752,-11.271,-45.057,179.855,5.862,149.088
C01515=1174.757,-11.521,-45.044,179.852,5.861,149.088
C01516=1174.762,-11.771,-45.031,179.849,5.861,149.089
C01517=1174.767,-12.020,-45.018,179.847,5.860,149.090
C01518=1174.773,-12.270,-45.005,179.845,5.859,149.090
C01519=1174.778,-12.520,-44.992,179.843,5.860,149.091
C01520=1174.783,-12.769,-44.980,179.840,5.859,149.091
C01521=1174.788,-13.018,-44.966,179.838,5.858,149.092
C01522=1174.793,-13.268,-44.953,179.835,5.858,149.093
C01523=1174.798,-13.518,-44.940,179.833,5.857,149.093
C01524=1174.804,-13.767,-44.927,179.830,5.857,149.094
C01525=1174.808,-14.017,-44.914,179.828,5.856,149.094
C01526=1174.814,-14.267,-44.901,179.825,5.855,149.095
C01527=1174.819,-14.516,-44.888,179.823,5.855,149.096
C01528=1174.824,-14.766,-44.875,179.821,5.854,149.096
C01529=1174.829,-15.015,-44.862,179.818,5.854,149.097
C01530=1174.834,-15.265,-44.850,179.815,5.853,149.098
C01531=1174.839,-15.515,-44.836,179.813,5.852,149.098
C01532=1174.845,-15.764,-44.824,179.810,5.852,149.099
C01533=1174.850,-16.014,-44.811,179.808,5.852,149.099
C01534=1174.855,-16.264,-44.798,179.806,5.851,149.100
C01535=1174.860,-16.513,-44.785,179.804,5.851,149.101
C01536=1174.865,-16.763,-44.772,179.801,5.851,149.101
C01537=1174.870,-17.013,-44.759,179.799,5.850,149.102
C01538=1174.876,-17.262,-44.746,179.796,5.849,149.103
C01539=1174.881,-17.512,-44.734,179.793,5.849,149.103
C01540=1174.886,-17.761,-44.721,179.791,5.848,149.104
C01541=1174.890,-18.011,-44.708,179.789,5.848,149.104
C01542=1174.896,-18.260,-44.695,179.786,5.847,149.105
C01543=1174.901,-18.510,-44.682,179.784,5.846,149.106
C01544=1174.907,-18.759,-44.670,179.781,5.846,149.106
C01545=1174.911,-19.009,-44.657,179.778,5.845,149.107
C01546=1174.916,-19.259,-44.644,179.776,5.845,149.107
C01547=1174.922,-19.509,-44.632,179.774,5.844,149.108
C01548=1174.927,-19.758,-44.619,179.772,5.844,149.109
C01549=1174.932,-20.008,-44.606,179.769,5.844,149.109
C01550=1174.937,-20.258,-44.593,179.767,5.843,149.110
C01551=1174.942,-20.507,-44.581,179.764,5.843,149.111
C01552=1174.947,-20.756,-44.568,179.762,5.842,149.111
C01553=1174.953,-21.006,-44.555,179.759,5.842,149.112
C01554=1174.958,-21.256,-44.543,179.757,5.841,149.112
C01555=1174.963,-21.506,-44.530,179.754,5.840,149.113
C01556=1174.968,-21.755,-44.518,179.752,5.840,149.114
C01557=1174.973,-22.005,-44.505,179.750,5.839,149.114
C01558=1174.978,-22.254,-44.492,179.747,5.839,149.115
C01559=1174.984,-22.504,-44.479,179.745,5.839,149.116
C01560=1174.989,-22.754,-44.467,179.743,5.838,149.116
C01561=1174.994,-23.003,-44.454,179.740,5.838,149.117
C01562=1174.999,-23.253,-44.441,179.737,5.837,149.117
C01563=1175.004,-23.522,-44.428,179.735,5.837,149.118
C01564=1175.011,-23.793,-44.414,179.732,5.836,149.119
C01565=1175.016,-24.063,-44.401,179.730,5.835,149.119
C01566=1175.021,-24.332,-44.387,179.727,5.835,149.120
C01567=1175.027,-24.582,-44.376,179.724,5.835,149.121
C01568=1175.031,-24.832,-44.363,179.722,5.834,149.121
C01569=1175.037,-25.081,-44.349,179.720,5.833,149.122
C01570=1175.042,-25.331,-44.337,179.717,5.833,149.122
C01571=1175.047,-25.581,-44.325,179.715,5.832,149.123
C01572=1175.053,-25.830,-44.312,179.712,5.832,149.124
C01573=1175.058,-26.079,-44.300,179.710,5.832,149.124
C01574=1175.063,-26.330,-44.288,179.708,5.831,149.125
C01575=1175.068,-26.579,-44.275,179.705,5.831,149.126
C01576=1175.073,-26.828,-44.262,179.703,5.830,149.126
C01577=1175.078,-27.078,-44.250,179.700,5.829,149.127
C01578=1175.083,-27.328,-44.238,179.698,5.829,149.127
C01579=1175.088,-27.577,-44.225,179.695,5.829,149.128
C01580=1175.094,-27.827,-44.213,179.693,5.828,149.129
C01581=1175.098,-28.077,-44.200,179.691,5.828,149.129
C01582=1175.104,-28.326,-44.188,179.688,5.828,149.130
C01583=1175.109,-28.576,-44.176,179.686,5.827,149.130
C01584=1175.114,-28.826,-44.163,179.683,5.826,149.131
C01585=1175.120,-29.076,-44.151,179.681,5.826,149.132
C01586=1175.125,-29.325,-44.139,179.678,5.825,149.132
C01587=1175.130,-29.574,-44.126,179.676,5.825,149.133
C01588=1175.135,-29.824,-44.114,179.673,5.824,149.134
C01589=1175.140,-30.073,-44.102,179.672,5.824,149.134
C01590=1175.145,-30.324,-44.089,179.669,5.824,149.135
C01591=1175.150,-30.573,-44.077,179.666,5.823,149.136
C01592=1175.156,-30.823,-44.065,179.664,5.823,149.136
C01593=1175.160,-31.072,-44.053,179.661,5.822,149.137
C01594=1175.166,-31.322,-44.041,179.659,5.822,149.137
C01595=1175.171,-31.572,-44.028,179.657,5.821,149.138
C01596=1175.176,-31.822,-44.017,179.654,5.821,149.139
C01597=1175.181,-32.071,-44.004,179.652,5.820,149.139
C01598=1175.187,-32.321,-43.992,179.650,5.820,149.140
C01599=1175.192,-32.570,-43.980,179.647,5.819,149.140
C01600=1175.197,-32.820,-43.968,179.645,5.819,149.141
C01601=1175.202,-33.069,-43.955,179.642,5.818,149.142
C01602=1175.208,-33.319,-43.943,179.640,5.819,149.142
C01603=1175.213,-33.569,-43.931,179.638,5.818,149.143
C01604=1175.218,-33.818,-43.919,179.635,5.817,149.143
C01605=1175.222,-34.068,-43.906,179.633,5.817,149.144
C01606=1175.228,-34.318,-43.894,179.630,5.816,149.145
C01607=1175.233,-34.567,-43.882,179.628,5.816,149.145
C01608=1175.238,-34.817,-43.870,179.625,5.815,149.146
C01609=1175.244,-35.067,-43.858,179.623,5.815,149.147
C01610=1175.249,-35.317,-43.845,179.621,5.815,149.147
C01611=1175.253,-35.566,-43.834,179.618,5.814,149.148
C01612=1175.258,-35.816,-43.822,179.616,5.814,149.148
C01613=1175.264,-36.066,-43.810,179.613,5.813,149.149
C01614=1175.269,-36.316,-43.798,179.611,5.812,149.150
C01615=1175.274,-36.565,-43.785,179.609,5.813,149.150
C01616=1175.280,-36.815,-43.773,179.606,5.812,149.151
C01617=1175.285,-37.064,-43.762,179.604,5.811,149.151
C01618=1175.290,-37.314,-43.749,179.602,5.811,149.152
C01619=1175.295,-37.564,-43.737,179.599,5.811,149.153
C01620=1175.301,-37.814,-43.726,179.597,5.810,149.153
C01621=1175.306,-38.063,-43.713,179.595,5.810,149.154
C01622=1175.310,-38.313,-43.702,179.592,5.810,149.155
C01623=1175.316,-38.562,-43.690,179.590,5.809,149.155
C01624=1175.321,-38.811,-43.678,179.587,5.808,149.156
C01625=1175.327,-39.061,-43.666,179.584,5.808,149.157
C01626=1175.332,-39.311,-43.654,179.583,5.808,149.157
C01627=1175.337,-39.561,-43.643,179.580,5.808,149.158
C01628=1175.342,-39.810,-43.630,179.578,5.807,149.158
C01629=1175.348,-40.060,-43.618,179.575,5.806,149.159
C01630=1175.352,-40.309,-43.607,179.573,5.806,149.160
C01631=1175.358,-40.559,-43.595,179.571,5.806,149.160
C01632=1175.363,-40.809,-43.582,179.568,5.805,149.161
C01633=1175.368,-41.059,-43.570,179.566,5.805,149.162
C01634=1175.373,-41.308,-43.559,179.564,5.804,149.162
C01635=1175.378,-41.558,-43.547,179.561,5.804,149.163
C01636=1175.384,-41.808,-43.535,179.558,5.803,149.163
C01637=1175.388,-42.057,-43.523,179.557,5.803,149.164
C01638=1175.394,-42.307,-43.511,179.554,5.803,149.165
C01639=1175.399,-42.557,-43.500,179.551,5.802,149.165
C01640=1175.404,-42.806,-43.489,179.549,5.802,149.166
C01641=1175.410,-43.056,-43.477,179.546,5.801,149.166
C01642=1175.415,-43.305,-43.464,179.544,5.802,149.167
C01643=1175.420,-43.555,-43.453,179.542,5.801,149.168
C01644=1175.425,-43.805,-43.441,179.540,5.800,149.168
C01645=1175.430,-44.055,-43.429,179.537,5.799,149.169
C01646=1175.435,-44.304,-43.418,179.535,5.800,149.169
C01647=1175.441,-44.554,-43.406,179.533,5.799,149.170
C01648=1175.446,-44.804,-43.394,179.530,5.799,149.171
C01649=1175.451,-45.054,-43.383,179.528,5.798,149.171
C01650=1175.456,-45.302,-43.371,179.525,5.798,149.172
C01651=1175.462,-45.552,-43.359,179.524,5.798,149.173
C01652=1175.467,-45.802,-43.347,179.521,5.797,149.173
C01653=1175.472,-46.052,-43.335,179.518,5.797,149.174
C01654=1175.477,-46.302,-43.324,179.516,5.796,149.174
C01655=1175.482,-46.551,-43.312,179.513,5.796,149.175
C01656=1175.488,-46.801,-43.300,179.512,5.796,149.176
C01657=1175.493,-47.050,-43.289,179.509,5.795,149.176
C01658=1175.498,-47.300,-43.278,179.506,5.795,149.177
C01659=1175.503,-47.550,-43.266,179.504,5.794,149.177
C01660=1175.508,-47.800,-43.254,179.502,5.794,149.178
C01661=1175.514,-48.050,-43.243,179.499,5.794,149.179
C01662=1175.519,-48.299,-43.231,179.497,5.793,149.179
C01663=1175.525,-48.549,-43.220,179.495,5.793,149.180
C01664=1175.529,-48.798,-43.208,179.492,5.792,149.181
C01665=1175.535,-49.048,-43.197,179.490,5.792,149.181
C01666=1175.539,-49.298,-43.185,179.488,5.792,149.182
C01667=1175.545,-49.567,-43.173,179.485,5.791,149.183
C01668=1175.551,-49.838,-43.160,179.483,5.791,149.183
C01669=1175.556,-50.109,-43.147,179.480,5.790,149.184
C01670=1175.562,-50.379,-43.136,179.478,5.790,149.185
C01671=1175.568,-50.629,-43.124,179.475,5.789,149.185
C01672=1175.573,-50.879,-43.112,179.473,5.789,149.186
C01673=1175.578,-51.129,-43.100,179.471,5.789,149.186
C01674=1175.583,-51.378,-43.089,179.468,5.788,149.187
C01675=1175.589,-51.627,-43.078,179.466,5.788,149.188
C01676=1175.593,-51.877,-43.066,179.464,5.788,149.188
C01677=1175.599,-52.127,-43.054,179.461,5.788,149.189
C01678=1175.604,-52.377,-43.044,179.459,5.787,149.189
C01679=1175.610,-52.626,-43.032,179.456,5.786,149.190
C01680=1175.615,-52.876,-43.021,179.455,5.786,149.191
C01681=1175.619,-53.126,-43.010,179.452,5.786,149.191
C01682=1175.625,-53.376,-42.998,179.449,5.786,149.192
C01683=1175.630,-53.625,-42.987,179.447,5.785,149.193
C01684=1175.635,-53.875,-42.975,179.445,5.785,149.193
C01685=1175.640,-54.125,-42.965,179.442,5.785,149.194
C01686=1175.646,-54.375,-42.953,179.440,5.784,149.194
C01687=1175.650,-54.624,-42.941,179.437,5.783,149.195
C01688=1175.656,-54.873,-42.930,179.436,5.783,149.196
C01689=1175.661,-55.123,-42.919,179.433,5.783,149.196
C01690=1175.666,-55.373,-42.907,179.431,5.783,149.197
C01691=1175.672,-55.623,-42.896,179.428,5.782,149.197
C01692=1175.677,-55.872,-42.885,179.426,5.782,149.198
C01693=1175.682,-56.122,-42.874,179.424,5.782,149.199
C01694=1175.687,-56.372,-42.862,179.421,5.781,149.199
C01695=1175.693,-56.621,-42.852,179.419,5.781,149.200
C01696=1175.698,-56.871,-42.840,179.417,5.781,149.201
C01697=1175.703,-57.121,-42.829,179.414,5.780,149.201
C01698=1175.707,-57.371,-42.817,179.412,5.780,149.202
C01699=1175.714,-57.620,-42.807,179.410,5.779,149.202
C01700=1175.718,-57.870,-42.795,179.408,5.779,149.203
C01701=1175.723,-58.120,-42.784,179.405,5.779,149.204
C01702=1175.729,-58.369,-42.772,179.403,5.778,149.204
C01703=1175.734,-58.619,-42.762,179.401,5.778,149.205
C01704=1175.739,-58.869,-42.751,179.398,5.778,149.206
C01705=1175.745,-59.118,-42.739,179.396,5.777,149.206
C01706=1175.750,-59.368,-42.728,179.393,5.777,149.207
C01707=1175.755,-59.618,-42.717,179.392,5.777,149.207
C01708=1175.761,-59.867,-42.706,179.389,5.776,149.208
C01709=1175.766,-60.117,-42.695,179.387,5.776,149.209
C01710=1175.770,-60.367,-42.684,179.384,5.775,149.209
C01711=1175.776,-60.616,-42.672,179.382,5.776,149.210
C01712=1175.781,-60.867,-42.662,179.380,5.775,149.210
C01713=1175.786,-61.116,-42.650,179.377,5.774,149.211
C01714=1175.791,-61.365,-42.639,179.375,5.775,149.212
C01715=1175.797,-61.616,-42.628,179.373,5.774,149.212
C01716=1175.802,-61.865,-42.617,179.370,5.774,149.213
C01717=1175.807,-62.115,-42.607,179.368,5.773,149.214
C01718=1175.812,-62.364,-42.596,179.366,5.773,149.214
C01719=1175.817,-62.614,-42.584,179.363,5.773,149.215
C01720=1175.823,-62.864,-42.573,179.361,5.772,149.215
C01721=1175.828,-63.114,-42.562,179.359,5.772,149.216
C01722=1175.833,-63.363,-42.552,179.357,5.771,149.217
C01723=1175.839,-63.613,-42.540,179.354,5.771,149.217
C01724=1175.844,-63.863,-42.529,179.351,5.771,149.218
C01725=1175.849,-64.112,-42.519,179.350,5.771,149.218
C01726=1175.854,-64.362,-42.507,179.347,5.770,149.219
C01727=1175.860,-64.612,-42.496,179.345,5.769,149.220
C01728=1175.865,-64.861,-42.485,179.343,5.770,149.220
C01729=1175.870,-65.112,-42.475,179.340,5.769,149.221
C01730=1175.875,-65.360,-42.464,179.338,5.769,149.222
C01731=1175.880,-65.611,-42.453,179.336,5.769,149.222
C01732=1175.886,-65.860,-42.442,179.334,5.768,149.223
C01733=1175.891,-66.110,-42.431,179.331,5.768,149.223
C01734=1175.896,-66.360,-42.420,179.328,5.767,149.224
C01735=1175.901,-66.609,-42.410,179.327,5.767,149.225
C01736=1175.906,-66.860,-42.399,179.324,5.767,149.225
C01737=1175.912,-67.108,-42.388,179.322,5.766,149.226
C01738=1175.917,-67.359,-42.377,179.320,5.767,149.227
C01739=1175.923,-67.608,-42.366,179.317,5.766,149.227
C01740=1175.928,-67.858,-42.355,179.315,5.765,149.228
C01741=1175.932,-68.108,-42.344,179.313,5.766,149.228
C01742=1175.938,-68.357,-42.334,179.311,5.765,149.229
C01743=1175.943,-68.607,-42.323,179.308,5.765,149.230
C01744=1175.949,-68.857,-42.312,179.306,5.765,149.230
C01745=1175.954,-69.107,-42.301,179.304,5.764,149.231
C01746=1175.959,-69.356,-42.290,179.301,5.764,149.232
C01747=1175.964,-69.606,-42.280,179.300,5.764,149.232
C01748=1175.970,-69.856,-42.269,179.297,5.763,149.233
C01749=1175.975,-70.105,-42.258,179.294,5.763,149.233
C01750=1175.980,-70.355,-42.248,179.292,5.762,149.234
C01751=1175.985,-70.605,-42.237,179.290,5.762,149.235
C01752=1175.991,-70.854,-42.226,179.288,5.762,149.235
C01753=1175.996,-71.105,-42.215,179.285,5.761,149.236
C01754=1176.002,-71.354,-42.204,179.284,5.761,149.236
C01755=1176.007,-71.604,-42.194,179.281,5.761,149.237
C01756=1176.012,-71.853,-42.184,179.278,5.760,149.238
C01757=1176.017,-72.103,-42.172,179.277,5.760,149.238
C01758=1176.022,-72.353,-42.162,179.274,5.760,149.239
C01759=1176.027,-72.603,-42.152,179.272,5.759,149.239
C01760=1176.033,-72.852,-42.141,179.270,5.760,149.240
C01761=1176.038,-73.102,-42.130,179.267,5.759,149.241
C01762=1176.043,-73.352,-42.120,179.265,5.758,149.241
C01763=1176.048,-73.602,-42.109,179.263,5.759,149.242
C01764=1176.054,-73.851,-42.098,179.261,5.758,149.242
C01765=1176.059,-74.101,-42.088,179.258,5.758,149.243
C01766=1176.064,-74.351,-42.078,179.256,5.758,149.244
C01767=1176.069,-74.601,-42.067,179.254,5.757,149.244
C01768=1176.074,-74.850,-42.056,179.251,5.757,149.245
C01769=1176.080,-75.099,-42.046,179.249,5.757,149.246
C01770=1176.085,-75.349,-42.035,179.247,5.756,149.246
C01771=1176.091,-75.621,-42.024,179.244,5.756,149.247
C01772=1176.097,-75.891,-42.012,179.242,5.755,149.247
C01773=1176.102,-76.163,-42.001,179.240,5.756,149.248
C01774=1176.108,-76.434,-41.989,179.237,5.755,149.249
C01775=1176.114,-76.684,-41.979,179.234,5.755,149.250
C01776=1176.119,-76.933,-41.968,179.233,5.755,149.250
C01777=1176.124,-77.183,-41.958,179.230,5.754,149.251
C01778=1176.130,-77.433,-41.947,179.228,5.754,149.251
C01779=1176.135,-77.683,-41.937,179.226,5.754,149.252
C01780=1176.140,-77.932,-41.927,179.224,5.753,149.252
C01781=1176.145,-78.182,-41.917,179.221,5.753,149.253
C01782=1176.150,-78.431,-41.906,179.219,5.753,149.254
C01783=1176.156,-78.681,-41.896,179.217,5.752,149.254
C01784=1176.161,-78.931,-41.885,179.214,5.752,149.255
C01785=1176.166,-79.180,-41.875,179.212,5.752,149.255
C01786=1176.172,-79.430,-41.865,179.210,5.752,149.256
C01787=1176.177,-79.680,-41.854,179.208,5.751,149.257
C01788=1176.182,-79.930,-41.844,179.205,5.751,149.257
C01789=1176.187,-80.180,-41.833,179.203,5.750,149.258
C01790=1176.193,-80.430,-41.823,179.201,5.751,149.259
C01791=1176.199,-80.679,-41.813,179.199,5.750,149.259
C01792=1176.203,-80.929,-41.801,179.196,5.750,149.260
C01793=1176.208,-81.178,-41.792,179.194,5.750,149.260
C01794=1176.213,-81.428,-41.781,179.192,5.749,149.261
C01795=1176.219,-81.678,-41.771,179.189,5.749,149.262
C01796=1176.224,-81.927,-41.761,179.188,5.749,149.262
C01797=1176.229,-82.178,-41.750,179.185,5.748,149.263
C01798=1176.235,-82.427,-41.740,179.182,5.748,149.264
C01799=1176.241,-82.677,-41.730,179.181,5.748,149.264
C01800=1176.245,-82.927,-41.720,179.178,5.748,149.265
C01801=1176.250,-83.176,-41.710,179.177,5.748,149.265
C01802=1176.256,-83.426,-41.699,179.174,5.747,149.266
C01803=1176.261,-83.676,-41.689,179.172,5.746,149.266
C01804=1176.267,-83.925,-41.679,179.170,5.747,149.267
C01805=1176.272,-84.175,-41.668,179.167,5.746,149.268
C01806=1176.276,-84.425,-41.659,179.165,5.746,149.268
C01807=1176.282,-84.675,-41.648,179.163,5.746,149.269
C01808=1176.288,-84.924,-41.638,179.161,5.745,149.270
C01809=1176.293,-85.174,-41.628,179.158,5.746,149.270
C01810=1176.298,-85.424,-41.617,179.156,5.745,149.271
C01811=1176.303,-85.673,-41.608,179.154,5.745,149.271
C01812=1176.308,-85.924,-41.598,179.152,5.745,149.272
C01813=1176.314,-86.173,-41.588,179.149,5.744,149.273
C01814=1176.320,-86.423,-41.577,179.147,5.743,149.273
C01815=1176.324,-86.673,-41.567,179.145,5.744,149.274
C01816=1176.329,-86.922,-41.557,179.143,5.743,149.274
C01817=1176.335,-87.172,-41.547,179.141,5.743,149.275
C01818=1176.341,-87.422,-41.537,179.139,5.743,149.275
C01819=1176.345,-87.672,-41.527,179.136,5.742,149.276
C01820=1176.350,-87.921,-41.517,179.134,5.743,149.277
C01821=1176.356,-88.171,-41.507,179.132,5.742,149.277
C01822=1176.361,-88.421,-41.497,179.130,5.742,149.278
C01823=1176.366,-88.671,-41.487,179.127,5.741,149.279
C01824=1176.372,-88.920,-41.477,179.125,5.741,149.279
